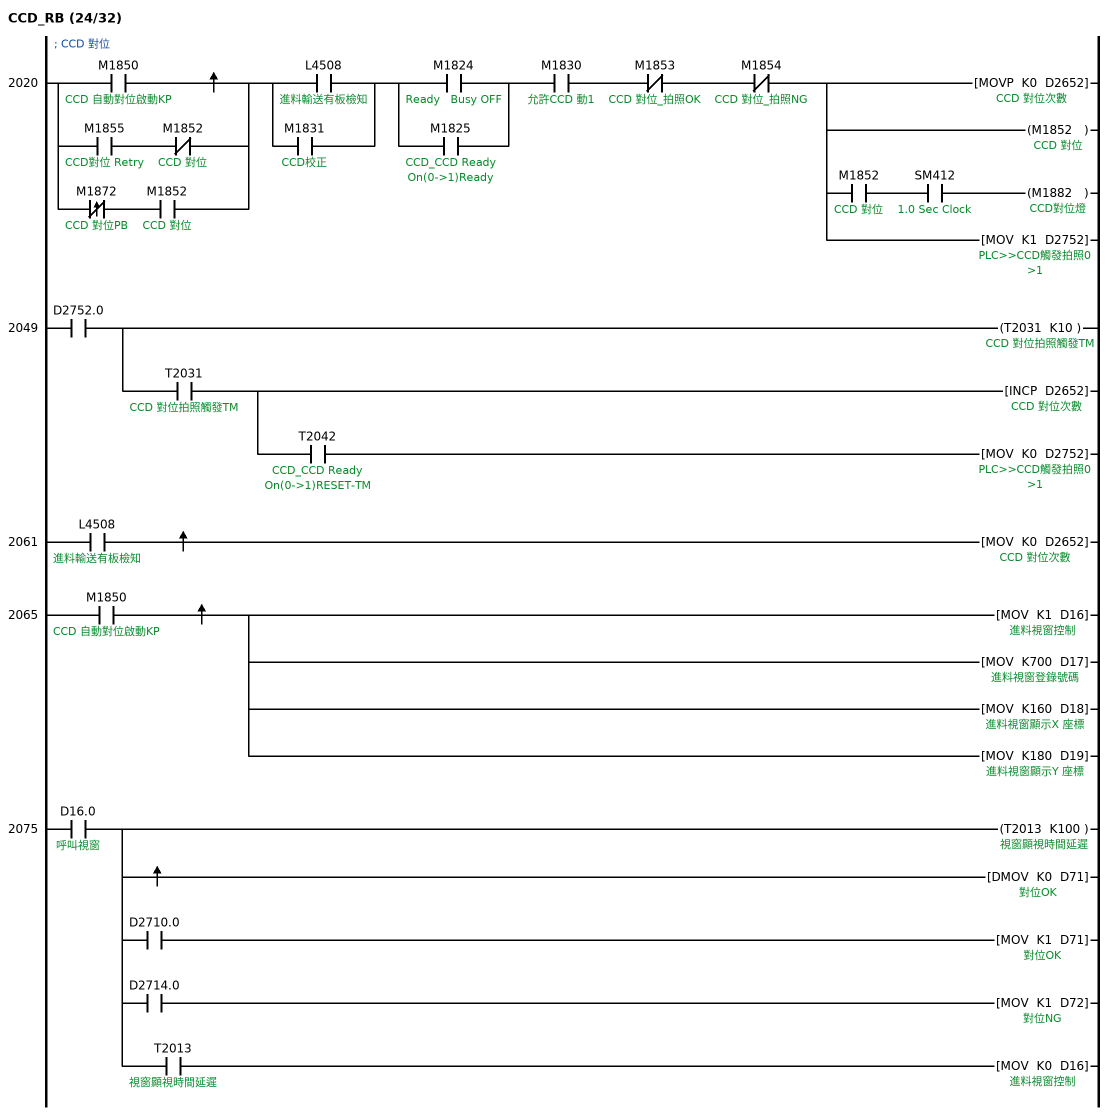
[picture p288: ladder of CCD_RB, rungs at steps 2020 to 2075]
; CCD 對位
2020  LD      M1850  ; CCD 自動對位啟動KP
      MEP
      LD      M1855  ; CCD對位 Retry
      ANI     M1852  ; CCD 對位
      ORB
      LDPI    M1872  ; CCD 對位PB
      AND     M1852  ; CCD 對位
      ORB
      LD      L4508  ; 進料輸送有板檢知
      OR      M1831  ; CCD校正
      ANB
      LD      M1824  ; Ready   Busy OFF
      OR      M1825  ; CCD_CCD Ready On(0->1)Ready
      ANB
      AND     M1830  ; 允許CCD 動1
      ANI     M1853  ; CCD 對位_拍照OK
      ANI     M1854  ; CCD 對位_拍照NG
      MOVP    K0 D2652  ; CCD 對位次數
      OUT     M1852  ; CCD 對位
      MPS
      AND     M1852  ; CCD 對位
      AND     SM412  ; 1.0 Sec Clock
      OUT     M1882  ; CCD對位燈
      MPP
      MOV     K1 D2752
2049  LD      D2752.0
      OUT     T2031 K10  ; CCD 對位拍照觸發TM
      AND     T2031  ; CCD 對位拍照觸發TM
      INCP    D2652
      AND     T2042  ; CCD_CCD Ready On(0->1)RESET-TM
      MOV     K0 D2752
2061  LD      L4508  ; 進料輸送有板檢知
      MEP
      MOV     K0 D2652
2065  LD      M1850  ; CCD 自動對位啟動KP
      MEP
      MOV     K1 D16  ; 進料視窗控制
      MOV     K700 D17  ; 進料視窗登錄號碼
      MOV     K160 D18  ; 進料視窗顯示X 座標
      MOV     K180 D19  ; 進料視窗顯示Y 座標
2075  LD      D16.0  ; 呼叫視窗
      OUT     T2013 K100  ; 視窗顯視時間延遲
      MPS
      MEP
      DMOV    K0 D71  ; 對位OK
      MRD
      AND     D2710.0
      MOV     K1 D71
      MRD
      AND     D2714.0
      MOV     K1 D72  ; 對位NG
      MPP
      AND     T2013  ; 視窗顯視時間延遲
      MOV     K0 D16
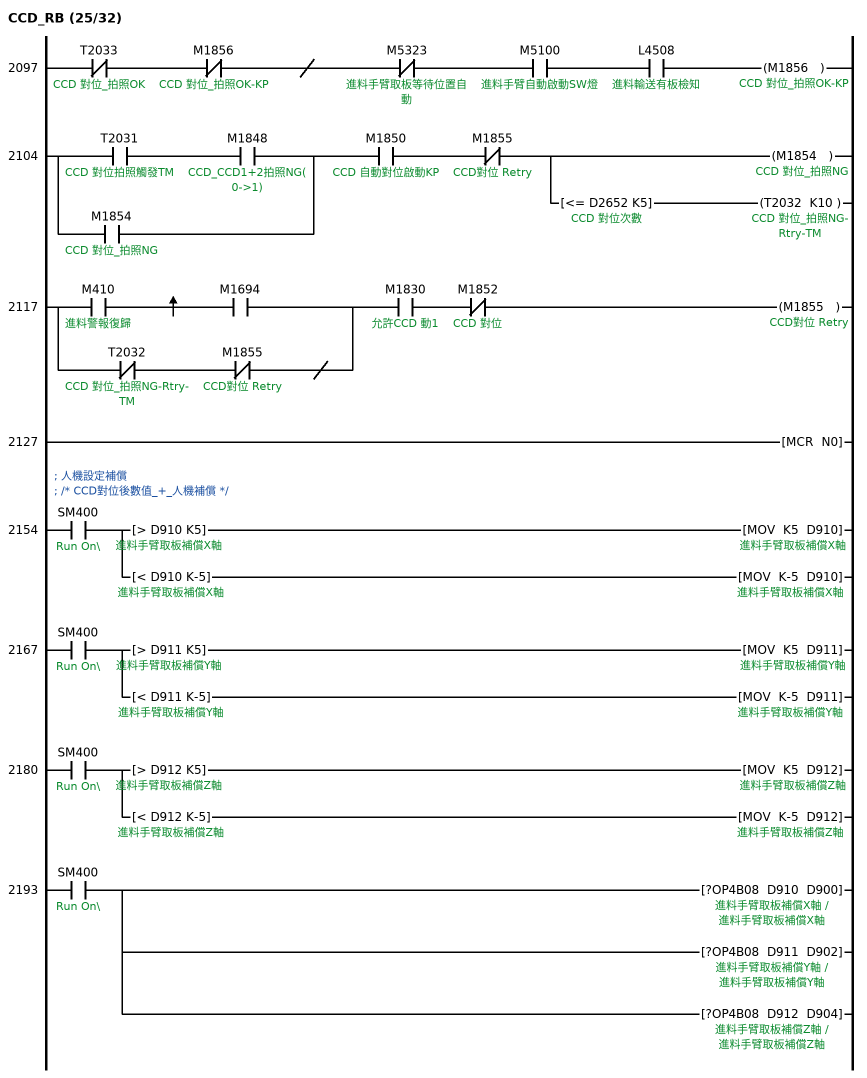
2097  LDI     T2033  ; CCD 對位_拍照OK
      ANI     M1856  ; CCD 對位_拍照OK-KP
      INV
      ANI     M5323  ; 進料手臂取板等待位置自動
      AND     M5100  ; 進料手臂自動啟動SW燈
      AND     L4508  ; 進料輸送有板檢知
      OUT     M1856  ; CCD 對位_拍照OK-KP
2104  LD      T2031  ; CCD 對位拍照觸發TM
      AND     M1848  ; CCD_CCD1+2拍照NG(0->1)
      OR      M1854  ; CCD 對位_拍照NG
      AND     M1850  ; CCD 自動對位啟動KP
      ANI     M1855  ; CCD對位 Retry
      OUT     M1854  ; CCD 對位_拍照NG
      AND<=   D2652 K5  ; CCD 對位次數
      OUT     T2032 K10  ; CCD 對位_拍照NG-Rtry-TM
2117  LD      M410  ; 進料警報復歸
      MEP
      AND     M1694
      LDI     T2032  ; CCD 對位_拍照NG-Rtry-TM
      ANI     M1855  ; CCD對位 Retry
      INV
      ORB
      AND     M1830  ; 允許CCD 動1
      ANI     M1852  ; CCD 對位
      OUT     M1855  ; CCD對位 Retry
2127  MCR     N0
; 人機設定補償
; /* CCD對位後數值_+_人機補償 */
2154  LD      SM400  ; Run On\
      MPS
      AND>    D910 K5  ; 進料手臂取板補償X軸
      MOV     K5 D910
      MPP
      AND<    D910 K-5  ; 進料手臂取板補償X軸
      MOV     K-5 D910
2167  LD      SM400  ; Run On\
      MPS
      AND>    D911 K5  ; 進料手臂取板補償Y軸
      MOV     K5 D911
      MPP
      AND<    D911 K-5  ; 進料手臂取板補償Y軸
      MOV     K-5 D911
2180  LD      SM400  ; Run On\
      MPS
      AND>    D912 K5  ; 進料手臂取板補償Z軸
      MOV     K5 D912
      MPP
      AND<    D912 K-5  ; 進料手臂取板補償Z軸
      MOV     K-5 D912
2193  LD      SM400  ; Run On\
      ?OP4B08 D910 D900  ; 進料手臂取板補償X軸
      ?OP4B08 D911 D902  ; 進料手臂取板補償Y軸
      ?OP4B08 D912 D904  ; 進料手臂取板補償Z軸
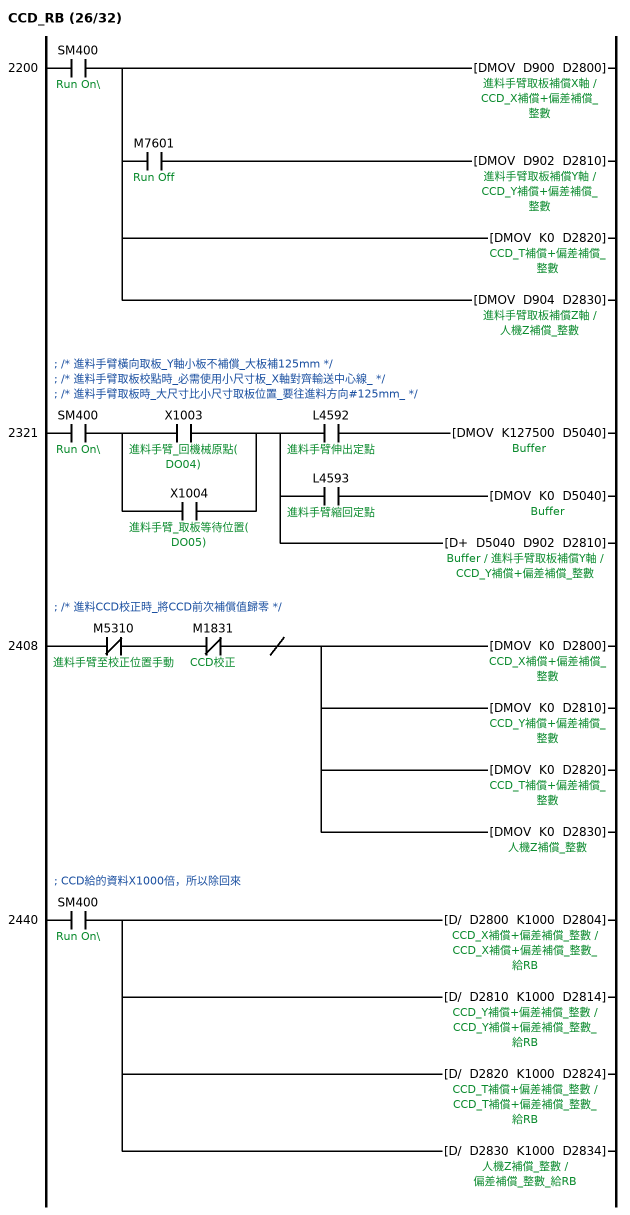
2200  LD      SM400  ; Run On\
      DMOV    D900 D2800  ; CCD_X補償+偏差補償_整數
      MPS
      AND     M7601  ; Run Off
      DMOV    D902 D2810  ; CCD_Y補償+偏差補償_整數
        [note] /* 在大/小板寬已補償位置_ */
      MPP
      DMOV    K0 D2820  ; CCD_T補償+偏差補償_整數
      DMOV    D904 D2830  ; 人機Z補償_整數
; /* 進料手臂橫向取板_Y軸小板不補償_大板補125mm */
; /* 進料手臂取板校點時_必需使用小尺寸板_X軸對齊輸送中心線_ */
; /* 進料手臂取板時_大尺寸比小尺寸取板位置_要往進料方向#125mm_ */
2321  LD      SM400  ; Run On\
      LD      X1003  ; 進料手臂_回機械原點(DO04)
      OR      X1004  ; 進料手臂_取板等待位置(DO05)
      ANB
      MPS
      AND     L4592  ; 進料手臂伸出定點
      DMOV    K127500 D5040  ; Buffer
        [note] /* 手臂大板寬_取板位_SHIFT */
      MRD
      AND     L4593  ; 進料手臂縮回定點
      DMOV    K0 D5040
        [note] /* 手臂大板寬_取板位_SHIFT */
      MPP
      D+      D5040 D902 D2810
        [note] /* 人機設定補正板長 */
; /* 進料CCD校正時_將CCD前次補償值歸零 */
2408  LDI     M5310  ; 進料手臂至校正位置手動
      ANI     M1831  ; CCD校正
      INV
      DMOV    K0 D2800
      DMOV    K0 D2810
      DMOV    K0 D2820
      DMOV    K0 D2830
; CCD給的資料X1000倍，所以除回來
2440  LD      SM400  ; Run On\
      D/      D2800 K1000 D2804
      D/      D2810 K1000 D2814
      D/      D2820 K1000 D2824
      D/      D2830 K1000 D2834  ; 偏差補償_整數_給RB
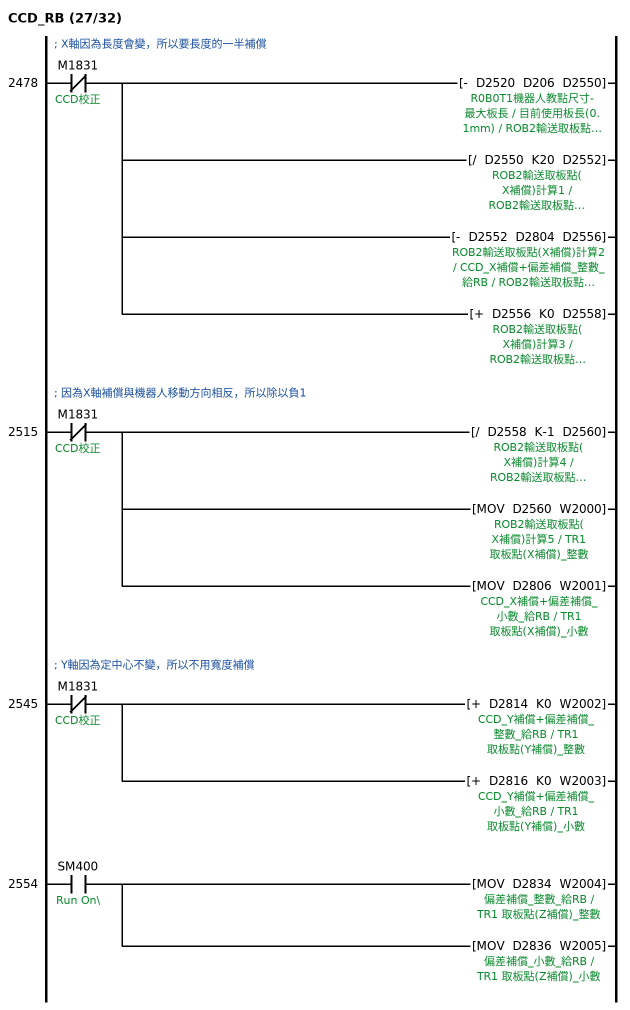
; X軸因為長度會變，所以要長度的一半補償
2478  LDI     M1831  ; CCD校正
      -       D2520 D206 D2550  ; R0B0T1機器人教點尺寸-最大板長 / 目前使用板長(0.1mm) / ROB2輸送取板點(X補償)計算1
      /       D2550 K20 D2552  ; ROB2輸送取板點(X補償)計算2
      -       D2552 D2804 D2556  ; ROB2輸送取板點(X補償)計算3
      +       D2556 K0 D2558  ; ROB2輸送取板點(X補償)計算4
; 因為X軸補償與機器人移動方向相反，所以除以負1
2515  LDI     M1831  ; CCD校正
      /       D2558 K-1 D2560  ; ROB2輸送取板點(X補償)計算5
      MOV     D2560 W2000  ; TR1 取板點(X補償)_整數
      MOV     D2806 W2001  ; CCD_X補償+偏差補償_小數_給RB / TR1 取板點(X補償)_小數
; Y軸因為定中心不變，所以不用寬度補償
2545  LDI     M1831  ; CCD校正
      +       D2814 K0 W2002  ; TR1 取板點(Y補償)_整數
      +       D2816 K0 W2003  ; CCD_Y補償+偏差補償_小數_給RB / TR1 取板點(Y補償)_小數
2554  LD      SM400  ; Run On\
      MOV     D2834 W2004  ; TR1 取板點(Z補償)_整數
      MOV     D2836 W2005  ; 偏差補償_小數_給RB / TR1 取板點(Z補償)_小數
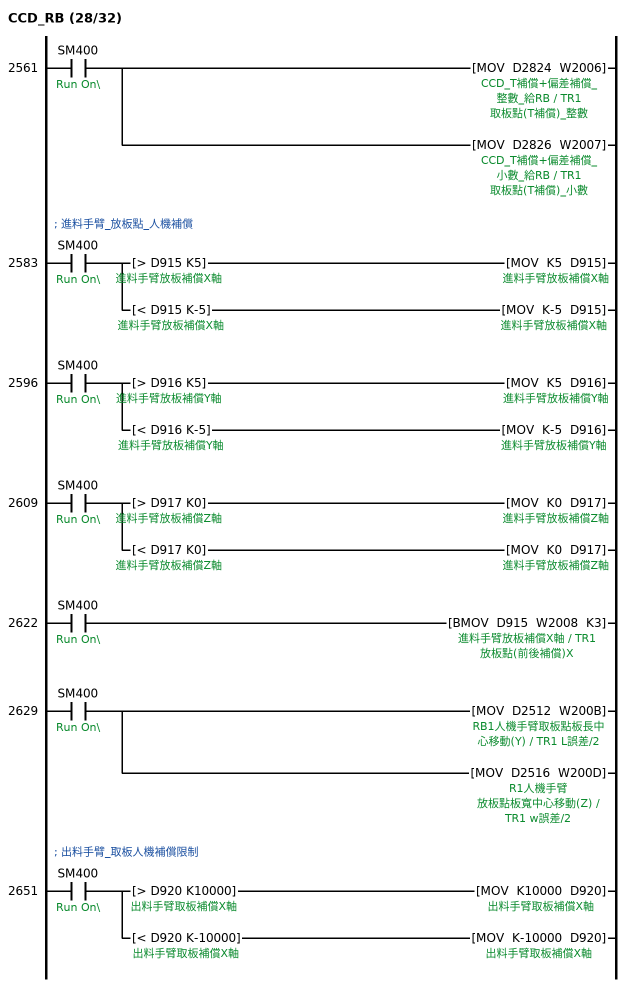
2561  LD      SM400  ; Run On\
      MOV     D2824 W2006  ; TR1 取板點(T補償)_整數
      MOV     D2826 W2007  ; CCD_T補償+偏差補償_小數_給RB / TR1 取板點(T補償)_小數
; 進料手臂_放板點_人機補償
2583  LD      SM400  ; Run On\
      MPS
      AND>    D915 K5  ; 進料手臂放板補償X軸
      MOV     K5 D915
      MPP
      AND<    D915 K-5  ; 進料手臂放板補償X軸
      MOV     K-5 D915
2596  LD      SM400  ; Run On\
      MPS
      AND>    D916 K5  ; 進料手臂放板補償Y軸
      MOV     K5 D916
      MPP
      AND<    D916 K-5  ; 進料手臂放板補償Y軸
      MOV     K-5 D916
2609  LD      SM400  ; Run On\
      MPS
      AND>    D917 K0  ; 進料手臂放板補償Z軸
      MOV     K0 D917
      MPP
      AND<    D917 K0  ; 進料手臂放板補償Z軸
      MOV     K0 D917
2622  LD      SM400  ; Run On\
      BMOV    D915 W2008 K3  ; TR1 放板點(前後補償)X
2629  LD      SM400  ; Run On\
      MOV     D2512 W200B  ; RB1人機手臂取板點板長中心移動(Y) / TR1 L誤差/2
      MOV     D2516 W200D  ; R1人機手臂 放板點板寬中心移動(Z) / TR1 w誤差/2
; 出料手臂_取板人機補償限制
2651  LD      SM400  ; Run On\
      MPS
      AND>    D920 K10000  ; 出料手臂取板補償X軸
      MOV     K10000 D920
      MPP
      AND<    D920 K-10000  ; 出料手臂取板補償X軸
      MOV     K-10000 D920
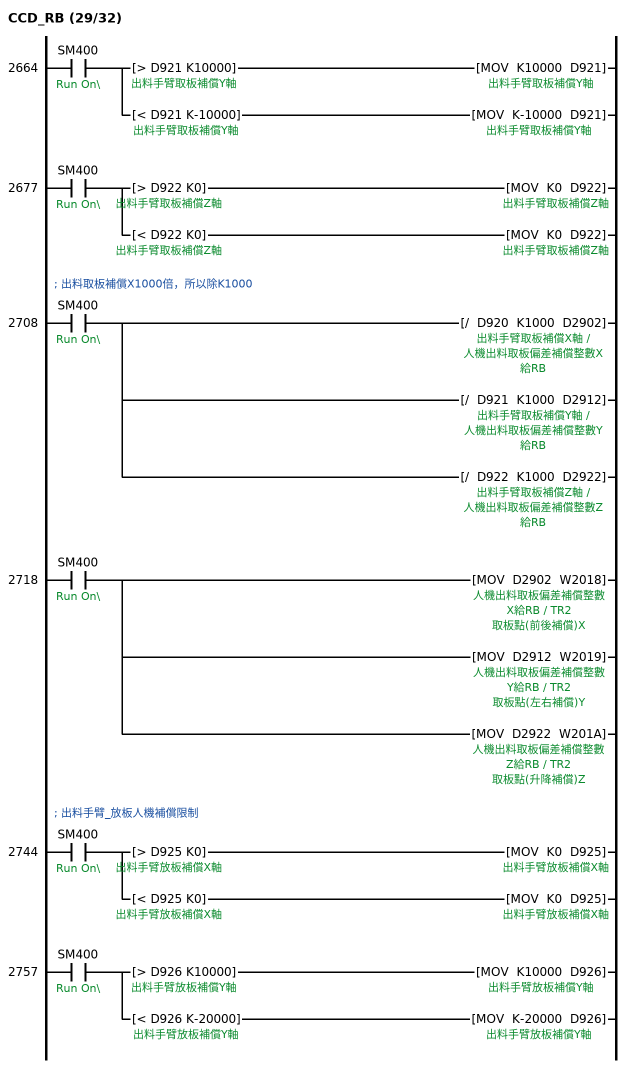
2664  LD      SM400  ; Run On\
      MPS
      AND>    D921 K10000  ; 出料手臂取板補償Y軸
      MOV     K10000 D921
      MPP
      AND<    D921 K-10000  ; 出料手臂取板補償Y軸
      MOV     K-10000 D921
2677  LD      SM400  ; Run On\
      MPS
      AND>    D922 K0  ; 出料手臂取板補償Z軸
      MOV     K0 D922
      MPP
      AND<    D922 K0  ; 出料手臂取板補償Z軸
      MOV     K0 D922
; 出料取板補償X1000倍，所以除K1000
2708  LD      SM400  ; Run On\
      /       D920 K1000 D2902  ; 人機出料取板偏差補償整數X給RB
      /       D921 K1000 D2912  ; 人機出料取板偏差補償整數Y給RB
      /       D922 K1000 D2922  ; 人機出料取板偏差補償整數Z給RB
2718  LD      SM400  ; Run On\
      MOV     D2902 W2018  ; TR2 取板點(前後補償)X
      MOV     D2912 W2019  ; TR2 取板點(左右補償)Y
      MOV     D2922 W201A  ; TR2 取板點(升降補償)Z
; 出料手臂_放板人機補償限制
2744  LD      SM400  ; Run On\
      MPS
      AND>    D925 K0  ; 出料手臂放板補償X軸
      MOV     K0 D925
      MPP
      AND<    D925 K0  ; 出料手臂放板補償X軸
      MOV     K0 D925
2757  LD      SM400  ; Run On\
      MPS
      AND>    D926 K10000  ; 出料手臂放板補償Y軸
      MOV     K10000 D926
      MPP
      AND<    D926 K-20000  ; 出料手臂放板補償Y軸
      MOV     K-20000 D926
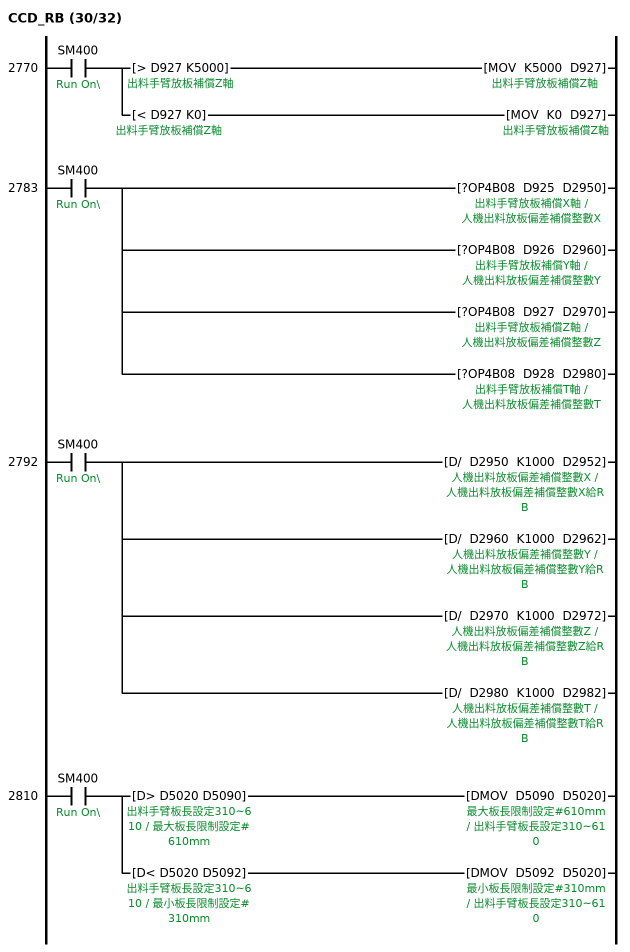
2770  LD      SM400  ; Run On\
      MPS
      AND>    D927 K5000  ; 出料手臂放板補償Z軸
      MOV     K5000 D927
      MPP
      AND<    D927 K0  ; 出料手臂放板補償Z軸
      MOV     K0 D927
2783  LD      SM400  ; Run On\
      ?OP4B08 D925 D2950  ; 人機出料放板偏差補償整數X
      ?OP4B08 D926 D2960  ; 人機出料放板偏差補償整數Y
      ?OP4B08 D927 D2970  ; 人機出料放板偏差補償整數Z
      ?OP4B08 D928 D2980  ; 出料手臂放板補償T軸 / 人機出料放板偏差補償整數T
2792  LD      SM400  ; Run On\
      D/      D2950 K1000 D2952  ; 人機出料放板偏差補償整數X給RB
      D/      D2960 K1000 D2962  ; 人機出料放板偏差補償整數Y給RB
      D/      D2970 K1000 D2972  ; 人機出料放板偏差補償整數Z給RB
      D/      D2980 K1000 D2982  ; 人機出料放板偏差補償整數T給RB
2810  LD      SM400  ; Run On\
      MPS
      ANDD>   D5020 D5090  ; 出料手臂板長設定310~610 / 最大板長限制設定#610mm
      DMOV    D5090 D5020
      MPP
      ANDD<   D5020 D5092  ; 出料手臂板長設定310~610 / 最小板長限制設定#310mm
      DMOV    D5092 D5020
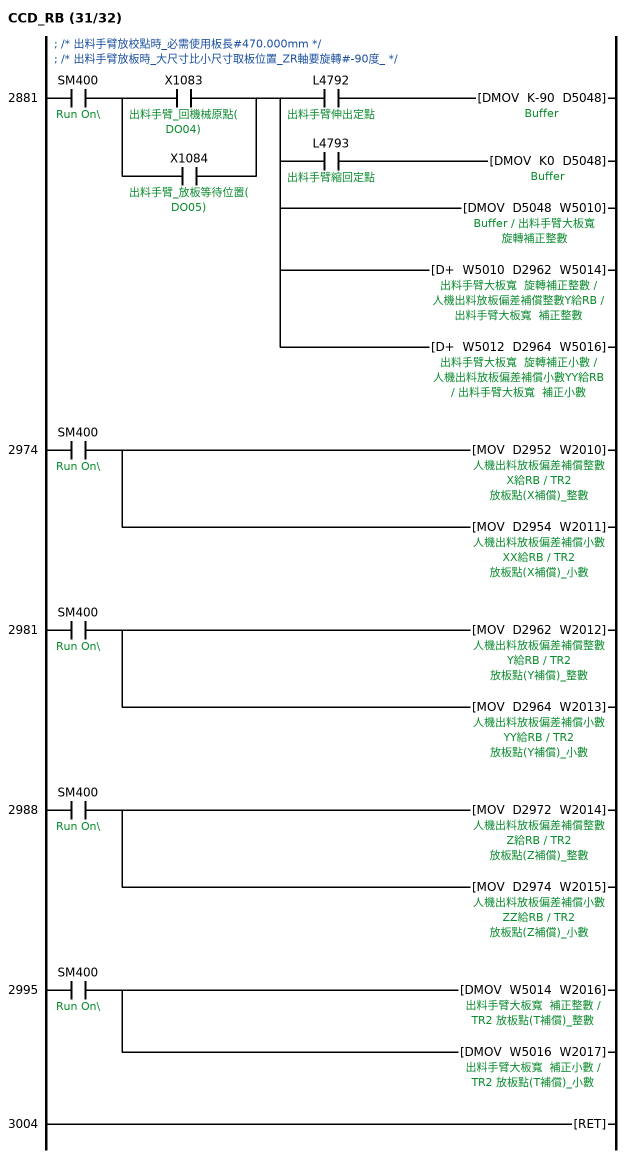
; /* 出料手臂放校點時_必需使用板長#470.000mm */
; /* 出料手臂放板時_大尺寸比小尺寸取板位置_ZR軸要旋轉#-90度_ */
2881  LD      SM400  ; Run On\
      LD      X1083  ; 出料手臂_回機械原點(DO04)
      OR      X1084  ; 出料手臂_放板等待位置(DO05)
      ANB
      MPS
      AND     L4792  ; 出料手臂伸出定點
      DMOV    K-90 D5048  ; Buffer
        [note] /* 手臂大板寬_取板位_SHIFT */
      MRD
      AND     L4793  ; 出料手臂縮回定點
      DMOV    K0 D5048
        [note] /* 手臂大板寬_取板位_SHIFT */
      MPP
      DMOV    D5048 W5010  ; 出料手臂大板寬  旋轉補正整數
      D+      W5010 D2962 W5014  ; 出料手臂大板寬  補正整數
        [note] /* 人機設定補正板長整數 */
      D+      W5012 D2964 W5016  ; 出料手臂大板寬  旋轉補正小數 / 人機出料放板偏差補償小數YY給RB / 出料手臂大板寬  補正小數
        [note] /* 人機設定補正板長小數 */
2974  LD      SM400  ; Run On\
      MOV     D2952 W2010  ; TR2 放板點(X補償)_整數
      MOV     D2954 W2011  ; 人機出料放板偏差補償小數XX給RB / TR2 放板點(X補償)_小數
2981  LD      SM400  ; Run On\
      MOV     D2962 W2012  ; TR2 放板點(Y補償)_整數
      MOV     D2964 W2013  ; TR2 放板點(Y補償)_小數
2988  LD      SM400  ; Run On\
      MOV     D2972 W2014  ; TR2 放板點(Z補償)_整數
      MOV     D2974 W2015  ; 人機出料放板偏差補償小數ZZ給RB / TR2 放板點(Z補償)_小數
2995  LD      SM400  ; Run On\
      DMOV    W5014 W2016  ; TR2 放板點(T補償)_整數
      DMOV    W5016 W2017  ; TR2 放板點(T補償)_小數
3004  RET
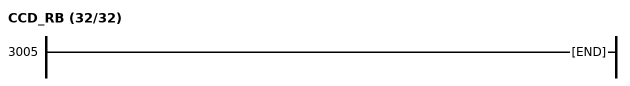
3005  END
END_PROGRAM

PROGRAM MECHA
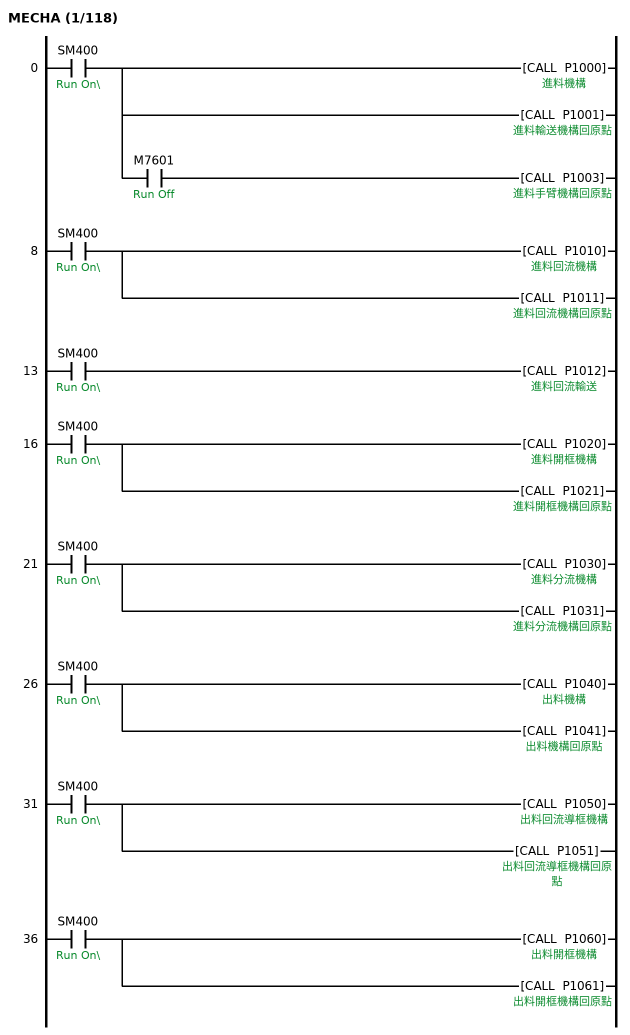
0     LD      SM400  ; Run On\
      CALL    P1000  ; 進料機構
      CALL    P1001  ; 進料輸送機構回原點
      AND     M7601  ; Run Off
      CALL    P1003  ; 進料手臂機構回原點
8     LD      SM400  ; Run On\
      CALL    P1010  ; 進料回流機構
      CALL    P1011  ; 進料回流機構回原點
13    LD      SM400  ; Run On\
      CALL    P1012  ; 進料回流輸送
16    LD      SM400  ; Run On\
      CALL    P1020  ; 進料開框機構
      CALL    P1021  ; 進料開框機構回原點
21    LD      SM400  ; Run On\
      CALL    P1030  ; 進料分流機構
      CALL    P1031  ; 進料分流機構回原點
26    LD      SM400  ; Run On\
      CALL    P1040  ; 出料機構
      CALL    P1041  ; 出料機構回原點
31    LD      SM400  ; Run On\
      CALL    P1050  ; 出料回流導框機構
      CALL    P1051  ; 出料回流導框機構回原點
36    LD      SM400  ; Run On\
      CALL    P1060  ; 出料開框機構
      CALL    P1061  ; 出料開框機構回原點
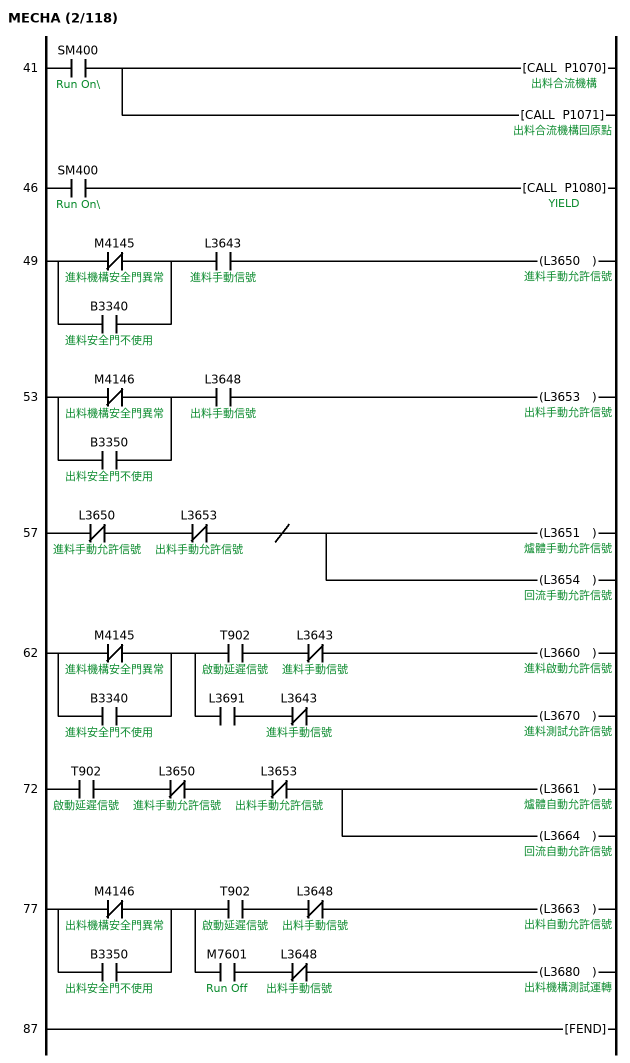
41    LD      SM400  ; Run On\
      CALL    P1070  ; 出料合流機構
      CALL    P1071  ; 出料合流機構回原點
46    LD      SM400  ; Run On\
      CALL    P1080  ; YIELD
49    LDI     M4145  ; 進料機構安全門異常
      OR      B3340  ; 進料安全門不使用
      AND     L3643  ; 進料手動信號
      OUT     L3650  ; 進料手動允許信號
53    LDI     M4146  ; 出料機構安全門異常
      OR      B3350  ; 出料安全門不使用
      AND     L3648  ; 出料手動信號
      OUT     L3653  ; 出料手動允許信號
57    LDI     L3650  ; 進料手動允許信號
      ANI     L3653  ; 出料手動允許信號
      INV
      OUT     L3651  ; 爐體手動允許信號
      OUT     L3654  ; 回流手動允許信號
62    LDI     M4145  ; 進料機構安全門異常
      OR      B3340  ; 進料安全門不使用
      MPS
      AND     T902  ; 啟動延遲信號
      ANI     L3643  ; 進料手動信號
      OUT     L3660  ; 進料啟動允許信號
      MPP
      AND     L3691
      ANI     L3643  ; 進料手動信號
      OUT     L3670  ; 進料測試允許信號
72    LD      T902  ; 啟動延遲信號
      ANI     L3650  ; 進料手動允許信號
      ANI     L3653  ; 出料手動允許信號
      OUT     L3661  ; 爐體自動允許信號
      OUT     L3664  ; 回流自動允許信號
77    LDI     M4146  ; 出料機構安全門異常
      OR      B3350  ; 出料安全門不使用
      MPS
      AND     T902  ; 啟動延遲信號
      ANI     L3648  ; 出料手動信號
      OUT     L3663  ; 出料自動允許信號
      MPP
      AND     M7601  ; Run Off
      ANI     L3648  ; 出料手動信號
      OUT     L3680  ; 出料機構測試運轉
87    FEND
; ---------進料機構------
      P1000
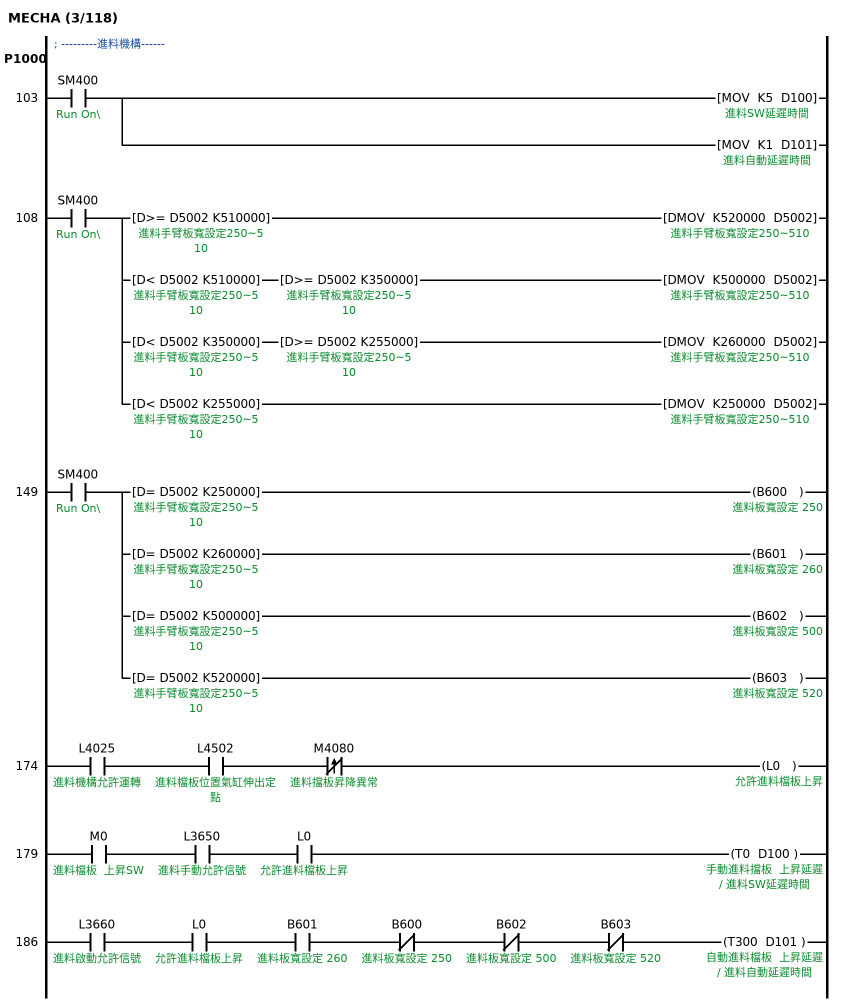
103   LD      SM400  ; Run On\
      MOV     K5 D100  ; 進料SW延遲時間
      MOV     K1 D101  ; 進料自動延遲時間
108   LD      SM400  ; Run On\
      MPS
      ANDD>=  D5002 K510000  ; 進料手臂板寬設定250~510
      DMOV    K520000 D5002
      MRD
      ANDD<   D5002 K510000  ; 進料手臂板寬設定250~510
      ANDD>=  D5002 K350000  ; 進料手臂板寬設定250~510
      DMOV    K500000 D5002
      MRD
      ANDD<   D5002 K350000  ; 進料手臂板寬設定250~510
      ANDD>=  D5002 K255000  ; 進料手臂板寬設定250~510
      DMOV    K260000 D5002
      MPP
      ANDD<   D5002 K255000  ; 進料手臂板寬設定250~510
      DMOV    K250000 D5002
149   LD      SM400  ; Run On\
      MPS
      ANDD=   D5002 K250000  ; 進料手臂板寬設定250~510
      OUT     B600  ; 進料板寬設定 250
      MRD
      ANDD=   D5002 K260000  ; 進料手臂板寬設定250~510
      OUT     B601  ; 進料板寬設定 260
      MRD
      ANDD=   D5002 K500000  ; 進料手臂板寬設定250~510
      OUT     B602  ; 進料板寬設定 500
      MPP
      ANDD=   D5002 K520000  ; 進料手臂板寬設定250~510
      OUT     B603  ; 進料板寬設定 520
174   LD      L4025  ; 進料機構允許運轉
      AND     L4502  ; 進料檔板位置氣缸伸出定點
      ANDPI   M4080  ; 進料擋板昇降異常
      OUT     L0  ; 允許進料檔板上昇
179   LD      M0  ; 進料檔板  上昇SW
      AND     L3650  ; 進料手動允許信號
      AND     L0  ; 允許進料檔板上昇
      OUT     T0 D100  ; 手動進料擋板  上昇延遲 / 進料SW延遲時間
186   LD      L3660  ; 進料啟動允許信號
      AND     L0  ; 允許進料檔板上昇
      AND     B601  ; 進料板寬設定 260
      ANI     B600  ; 進料板寬設定 250
      ANI     B602  ; 進料板寬設定 500
      ANI     B603  ; 進料板寬設定 520
      OUT     T300 D101  ; 自動進料檔板  上昇延遲 / 進料自動延遲時間
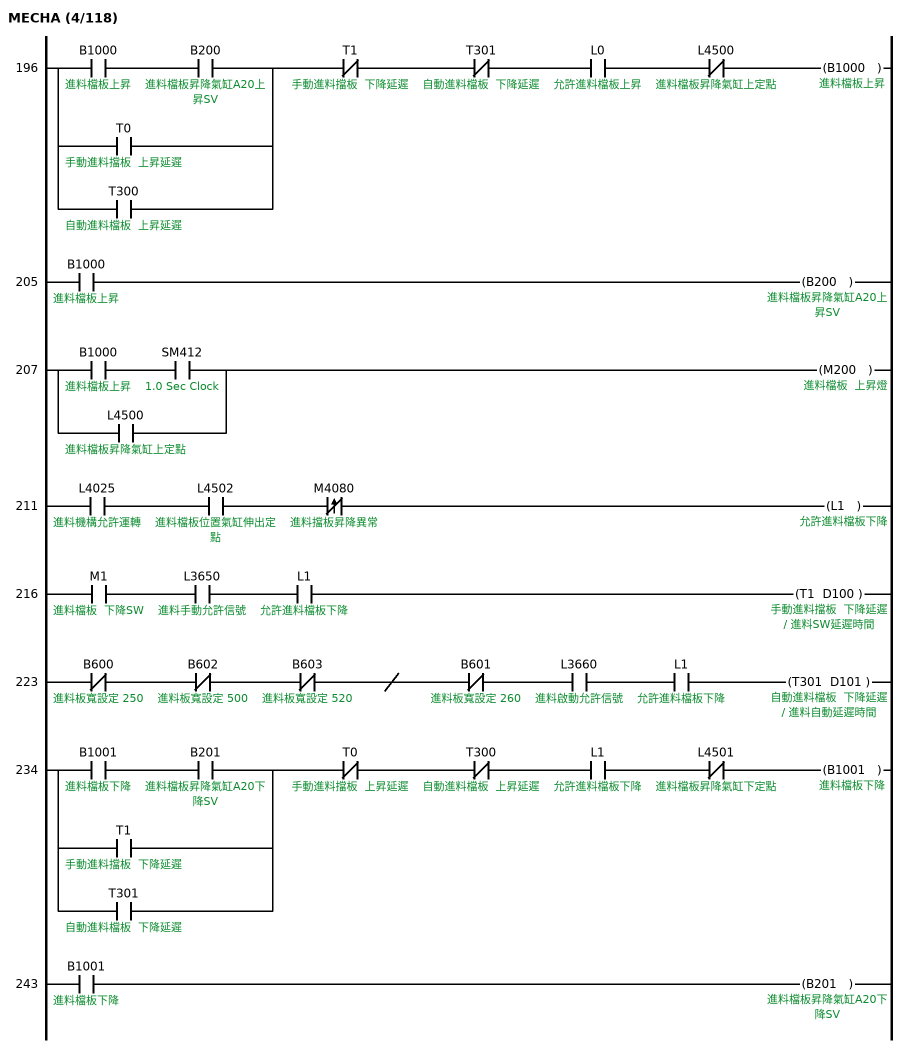
196   LD      B1000  ; 進料檔板上昇
      AND     B200  ; 進料檔板昇降氣缸A20上昇SV
      OR      T0  ; 手動進料擋板  上昇延遲
      OR      T300  ; 自動進料檔板  上昇延遲
      ANI     T1  ; 手動進料擋板  下降延遲
      ANI     T301  ; 自動進料檔板  下降延遲
      AND     L0  ; 允許進料檔板上昇
      ANI     L4500  ; 進料檔板昇降氣缸上定點
      OUT     B1000  ; 進料檔板上昇
205   LD      B1000  ; 進料檔板上昇
      OUT     B200  ; 進料檔板昇降氣缸A20上昇SV
207   LD      B1000  ; 進料檔板上昇
      AND     SM412  ; 1.0 Sec Clock
      OR      L4500  ; 進料檔板昇降氣缸上定點
      OUT     M200  ; 進料檔板  上昇燈
211   LD      L4025  ; 進料機構允許運轉
      AND     L4502  ; 進料檔板位置氣缸伸出定點
      ANDPI   M4080  ; 進料擋板昇降異常
      OUT     L1  ; 允許進料檔板下降
216   LD      M1  ; 進料檔板  下降SW
      AND     L3650  ; 進料手動允許信號
      AND     L1  ; 允許進料檔板下降
      OUT     T1 D100  ; 手動進料擋板  下降延遲 / 進料SW延遲時間
223   LDI     B600  ; 進料板寬設定 250
      ANI     B602  ; 進料板寬設定 500
      ANI     B603  ; 進料板寬設定 520
      INV
      ANI     B601  ; 進料板寬設定 260
      AND     L3660  ; 進料啟動允許信號
      AND     L1  ; 允許進料檔板下降
      OUT     T301 D101  ; 自動進料檔板  下降延遲 / 進料自動延遲時間
234   LD      B1001  ; 進料檔板下降
      AND     B201  ; 進料檔板昇降氣缸A20下降SV
      OR      T1  ; 手動進料擋板  下降延遲
      OR      T301  ; 自動進料檔板  下降延遲
      ANI     T0  ; 手動進料擋板  上昇延遲
      ANI     T300  ; 自動進料檔板  上昇延遲
      AND     L1  ; 允許進料檔板下降
      ANI     L4501  ; 進料檔板昇降氣缸下定點
      OUT     B1001  ; 進料檔板下降
243   LD      B1001  ; 進料檔板下降
      OUT     B201  ; 進料檔板昇降氣缸A20下降SV
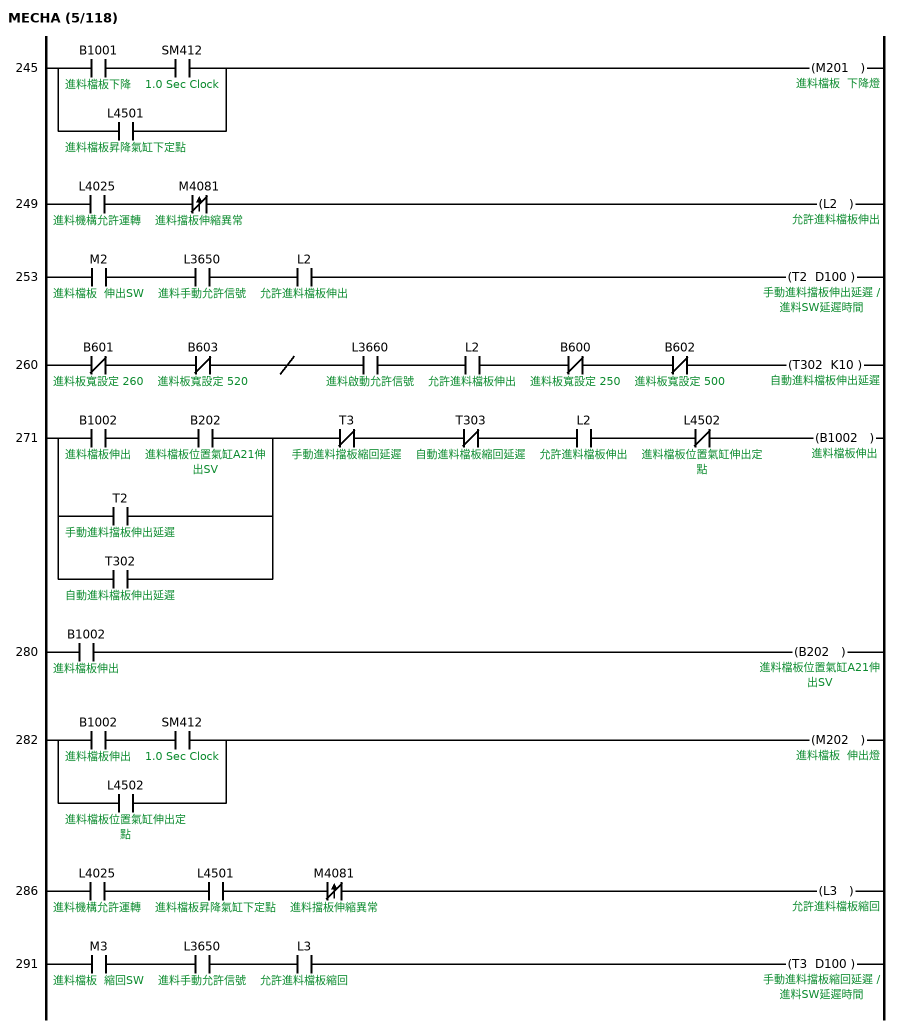
245   LD      B1001  ; 進料檔板下降
      AND     SM412  ; 1.0 Sec Clock
      OR      L4501  ; 進料檔板昇降氣缸下定點
      OUT     M201  ; 進料檔板  下降燈
249   LD      L4025  ; 進料機構允許運轉
      ANDPI   M4081  ; 進料擋板伸縮異常
      OUT     L2  ; 允許進料檔板伸出
253   LD      M2  ; 進料檔板  伸出SW
      AND     L3650  ; 進料手動允許信號
      AND     L2  ; 允許進料檔板伸出
      OUT     T2 D100  ; 手動進料擋板伸出延遲 / 進料SW延遲時間
260   LDI     B601  ; 進料板寬設定 260
      ANI     B603  ; 進料板寬設定 520
      INV
      AND     L3660  ; 進料啟動允許信號
      AND     L2  ; 允許進料檔板伸出
      ANI     B600  ; 進料板寬設定 250
      ANI     B602  ; 進料板寬設定 500
      OUT     T302 K10  ; 自動進料檔板伸出延遲
271   LD      B1002  ; 進料檔板伸出
      AND     B202  ; 進料檔板位置氣缸A21伸出SV
      OR      T2  ; 手動進料擋板伸出延遲
      OR      T302  ; 自動進料檔板伸出延遲
      ANI     T3  ; 手動進料擋板縮回延遲
      ANI     T303  ; 自動進料檔板縮回延遲
      AND     L2  ; 允許進料檔板伸出
      ANI     L4502  ; 進料檔板位置氣缸伸出定點
      OUT     B1002  ; 進料檔板伸出
280   LD      B1002  ; 進料檔板伸出
      OUT     B202  ; 進料檔板位置氣缸A21伸出SV
282   LD      B1002  ; 進料檔板伸出
      AND     SM412  ; 1.0 Sec Clock
      OR      L4502  ; 進料檔板位置氣缸伸出定點
      OUT     M202  ; 進料檔板  伸出燈
286   LD      L4025  ; 進料機構允許運轉
      AND     L4501  ; 進料檔板昇降氣缸下定點
      ANDPI   M4081  ; 進料擋板伸縮異常
      OUT     L3  ; 允許進料檔板縮回
291   LD      M3  ; 進料檔板  縮回SW
      AND     L3650  ; 進料手動允許信號
      AND     L3  ; 允許進料檔板縮回
      OUT     T3 D100  ; 手動進料擋板縮回延遲 / 進料SW延遲時間
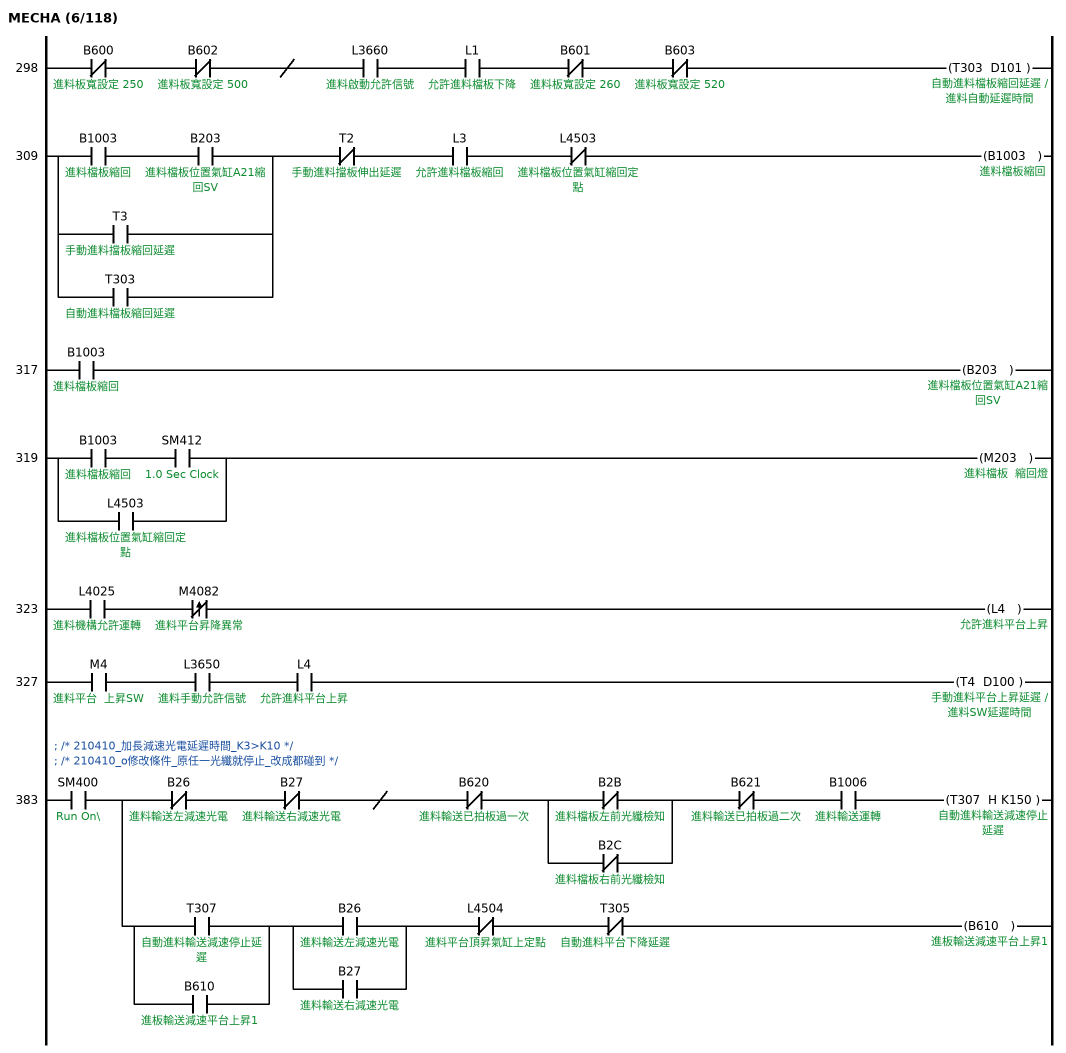
298   LDI     B600  ; 進料板寬設定 250
      ANI     B602  ; 進料板寬設定 500
      INV
      AND     L3660  ; 進料啟動允許信號
      AND     L1  ; 允許進料檔板下降
      ANI     B601  ; 進料板寬設定 260
      ANI     B603  ; 進料板寬設定 520
      OUT     T303 D101  ; 自動進料檔板縮回延遲 / 進料自動延遲時間
309   LD      B1003  ; 進料檔板縮回
      AND     B203  ; 進料檔板位置氣缸A21縮回SV
      OR      T3  ; 手動進料擋板縮回延遲
      OR      T303  ; 自動進料檔板縮回延遲
      ANI     T2  ; 手動進料擋板伸出延遲
      AND     L3  ; 允許進料檔板縮回
      ANI     L4503  ; 進料檔板位置氣缸縮回定點
      OUT     B1003  ; 進料檔板縮回
317   LD      B1003  ; 進料檔板縮回
      OUT     B203  ; 進料檔板位置氣缸A21縮回SV
319   LD      B1003  ; 進料檔板縮回
      AND     SM412  ; 1.0 Sec Clock
      OR      L4503  ; 進料檔板位置氣缸縮回定點
      OUT     M203  ; 進料檔板  縮回燈
323   LD      L4025  ; 進料機構允許運轉
      ANDPI   M4082  ; 進料平台昇降異常
      OUT     L4  ; 允許進料平台上昇
327   LD      M4  ; 進料平台  上昇SW
      AND     L3650  ; 進料手動允許信號
      AND     L4  ; 允許進料平台上昇
      OUT     T4 D100  ; 手動進料平台上昇延遲 / 進料SW延遲時間
; /* 210410_加長減速光電延遲時間_K3>K10 */
; /* 210410_o修改條件_原任一光纖就停止_改成都碰到 */
383   LD      SM400  ; Run On\
      MPS
      ANI     B26  ; 進料輸送左減速光電
      ANI     B27  ; 進料輸送右減速光電
      INV
      ANI     B620  ; 進料輸送已拍板過一次
      LDI     B2B  ; 進料檔板左前光纖檢知
      ORI     B2C  ; 進料檔板右前光纖檢知
      ANB
      ANI     B621  ; 進料輸送已拍板過二次
      AND     B1006  ; 進料輸送運轉
      OUTH    T307 K150  ; 自動進料輸送減速停止延遲
      MPP
      LD      T307  ; 自動進料輸送減速停止延遲
      OR      B610  ; 進板輸送減速平台上昇1
      ANB
      LD      B26  ; 進料輸送左減速光電
      OR      B27  ; 進料輸送右減速光電
      ANB
      ANI     L4504  ; 進料平台頂昇氣缸上定點
      ANI     T305  ; 自動進料平台下降延遲
      OUT     B610  ; 進板輸送減速平台上昇1
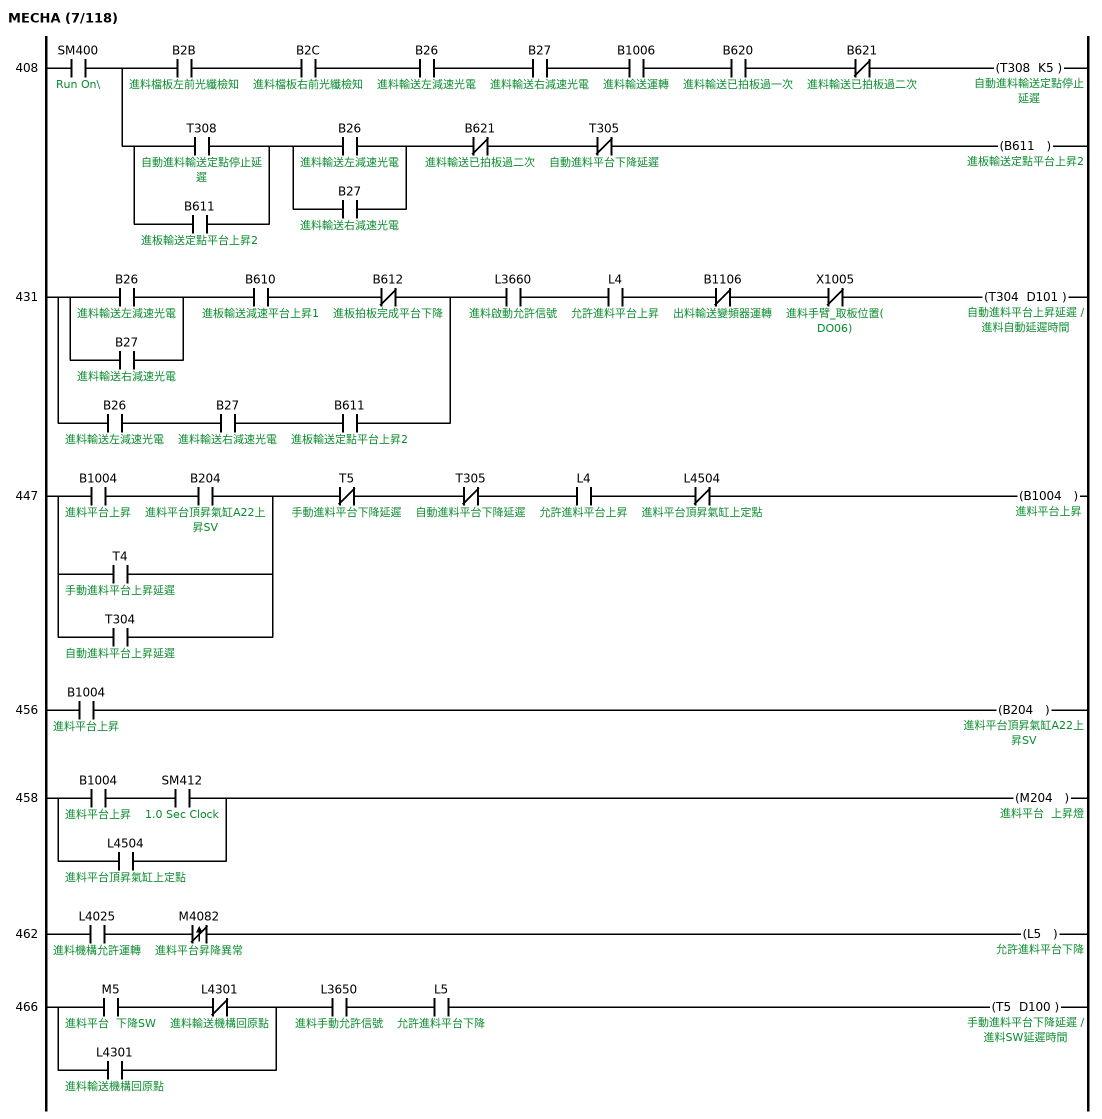
408   LD      SM400  ; Run On\
      MPS
      AND     B2B  ; 進料檔板左前光纖檢知
      AND     B2C  ; 進料檔板右前光纖檢知
      AND     B26  ; 進料輸送左減速光電
      AND     B27  ; 進料輸送右減速光電
      AND     B1006  ; 進料輸送運轉
      AND     B620  ; 進料輸送已拍板過一次
      ANI     B621  ; 進料輸送已拍板過二次
      OUT     T308 K5  ; 自動進料輸送定點停止延遲
      MPP
      LD      T308  ; 自動進料輸送定點停止延遲
      OR      B611  ; 進板輸送定點平台上昇2
      ANB
      LD      B26  ; 進料輸送左減速光電
      OR      B27  ; 進料輸送右減速光電
      ANB
      ANI     B621  ; 進料輸送已拍板過二次
      ANI     T305  ; 自動進料平台下降延遲
      OUT     B611  ; 進板輸送定點平台上昇2
431   LD      B26  ; 進料輸送左減速光電
      OR      B27  ; 進料輸送右減速光電
      AND     B610  ; 進板輸送減速平台上昇1
      ANI     B612  ; 進板拍板完成平台下降
      LD      B26  ; 進料輸送左減速光電
      AND     B27  ; 進料輸送右減速光電
      AND     B611  ; 進板輸送定點平台上昇2
      ORB
      AND     L3660  ; 進料啟動允許信號
      AND     L4  ; 允許進料平台上昇
      ANI     B1106  ; 出料輸送變頻器運轉
      ANI     X1005  ; 進料手臂_取板位置(DO06)
      OUT     T304 D101  ; 自動進料平台上昇延遲 / 進料自動延遲時間
447   LD      B1004  ; 進料平台上昇
      AND     B204  ; 進料平台頂昇氣缸A22上昇SV
      OR      T4  ; 手動進料平台上昇延遲
      OR      T304  ; 自動進料平台上昇延遲
      ANI     T5  ; 手動進料平台下降延遲
      ANI     T305  ; 自動進料平台下降延遲
      AND     L4  ; 允許進料平台上昇
      ANI     L4504  ; 進料平台頂昇氣缸上定點
      OUT     B1004  ; 進料平台上昇
456   LD      B1004  ; 進料平台上昇
      OUT     B204  ; 進料平台頂昇氣缸A22上昇SV
458   LD      B1004  ; 進料平台上昇
      AND     SM412  ; 1.0 Sec Clock
      OR      L4504  ; 進料平台頂昇氣缸上定點
      OUT     M204  ; 進料平台  上昇燈
462   LD      L4025  ; 進料機構允許運轉
      ANDPI   M4082  ; 進料平台昇降異常
      OUT     L5  ; 允許進料平台下降
466   LD      M5  ; 進料平台  下降SW
      ANI     L4301  ; 進料輸送機構回原點
      OR      L4301  ; 進料輸送機構回原點
      AND     L3650  ; 進料手動允許信號
      AND     L5  ; 允許進料平台下降
      OUT     T5 D100  ; 手動進料平台下降延遲 / 進料SW延遲時間
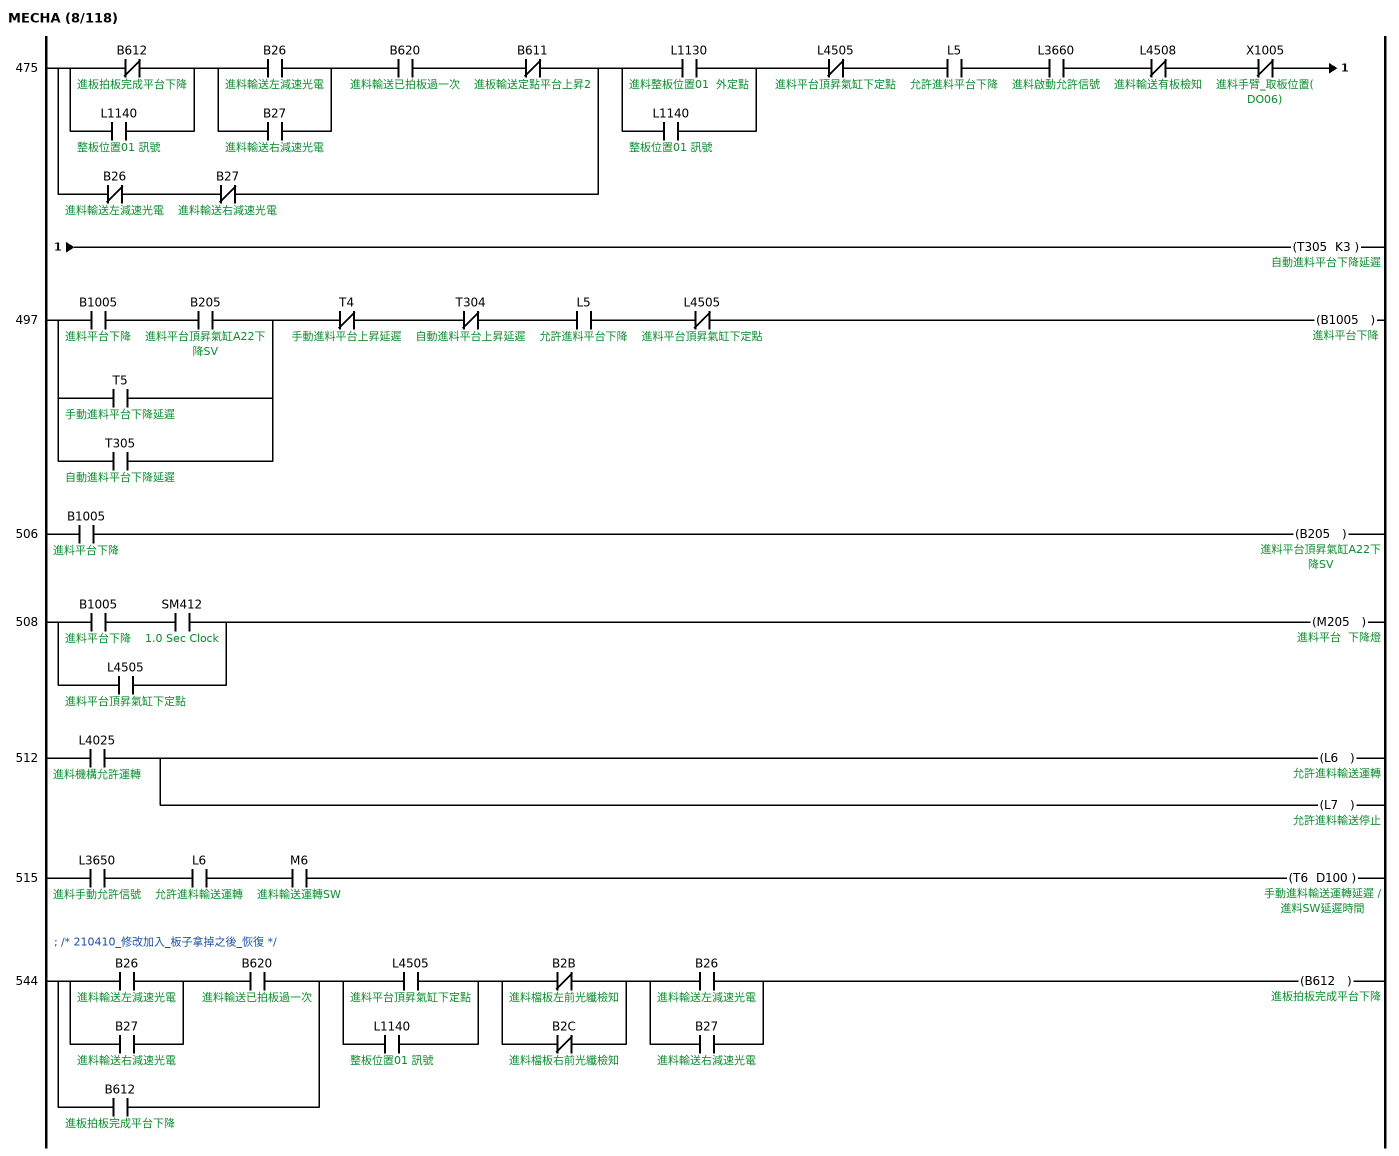
475   LDI     B612  ; 進板拍板完成平台下降
      OR      L1140  ; 整板位置01 訊號
      LD      B26  ; 進料輸送左減速光電
      OR      B27  ; 進料輸送右減速光電
      ANB
      AND     B620  ; 進料輸送已拍板過一次
      ANI     B611  ; 進板輸送定點平台上昇2
      LDI     B26  ; 進料輸送左減速光電
      ANI     B27  ; 進料輸送右減速光電
      ORB
      LD      L1130  ; 進料整板位置01  外定點
      OR      L1140  ; 整板位置01 訊號
      ANB
      ANI     L4505  ; 進料平台頂昇氣缸下定點
      AND     L5  ; 允許進料平台下降
      AND     L3660  ; 進料啟動允許信號
      ANI     L4508  ; 進料輸送有板檢知
      ANI     X1005  ; 進料手臂_取板位置(DO06)
      OUT     T305 K3  ; 自動進料平台下降延遲
497   LD      B1005  ; 進料平台下降
      AND     B205  ; 進料平台頂昇氣缸A22下降SV
      OR      T5  ; 手動進料平台下降延遲
      OR      T305  ; 自動進料平台下降延遲
      ANI     T4  ; 手動進料平台上昇延遲
      ANI     T304  ; 自動進料平台上昇延遲
      AND     L5  ; 允許進料平台下降
      ANI     L4505  ; 進料平台頂昇氣缸下定點
      OUT     B1005  ; 進料平台下降
506   LD      B1005  ; 進料平台下降
      OUT     B205  ; 進料平台頂昇氣缸A22下降SV
508   LD      B1005  ; 進料平台下降
      AND     SM412  ; 1.0 Sec Clock
      OR      L4505  ; 進料平台頂昇氣缸下定點
      OUT     M205  ; 進料平台  下降燈
512   LD      L4025  ; 進料機構允許運轉
      OUT     L6  ; 允許進料輸送運轉
      OUT     L7  ; 允許進料輸送停止
515   LD      L3650  ; 進料手動允許信號
      AND     L6  ; 允許進料輸送運轉
      AND     M6  ; 進料輸送運轉SW
      OUT     T6 D100  ; 手動進料輸送運轉延遲 / 進料SW延遲時間
; /* 210410_修改加入_板子拿掉之後_恢復 */
544   LD      B26  ; 進料輸送左減速光電
      OR      B27  ; 進料輸送右減速光電
      AND     B620  ; 進料輸送已拍板過一次
      OR      B612  ; 進板拍板完成平台下降
      LD      L4505  ; 進料平台頂昇氣缸下定點
      OR      L1140  ; 整板位置01 訊號
      ANB
      LDI     B2B  ; 進料檔板左前光纖檢知
      ORI     B2C  ; 進料檔板右前光纖檢知
      ANB
      LD      B26  ; 進料輸送左減速光電
      OR      B27  ; 進料輸送右減速光電
      ANB
      OUT     B612  ; 進板拍板完成平台下降
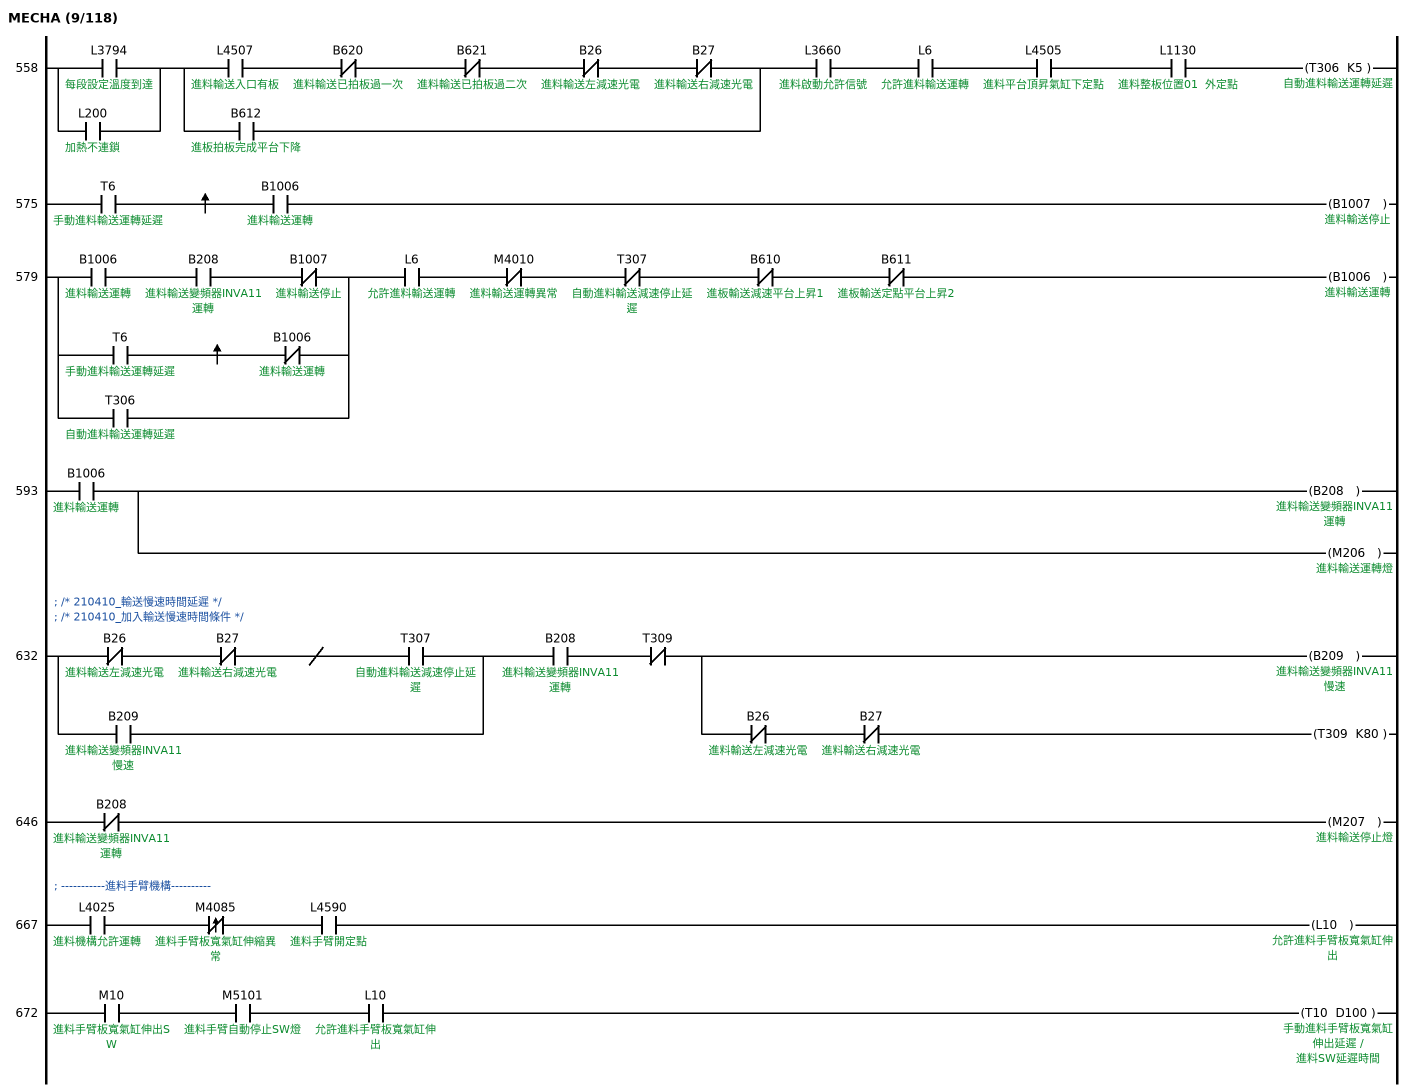
558   LD      L3794  ; 每段設定溫度到達
      OR      L200  ; 加熱不連鎖
      LD      L4507  ; 進料輸送入口有板
      ANI     B620  ; 進料輸送已拍板過一次
      ANI     B621  ; 進料輸送已拍板過二次
      ANI     B26  ; 進料輸送左減速光電
      ANI     B27  ; 進料輸送右減速光電
      OR      B612  ; 進板拍板完成平台下降
      ANB
      AND     L3660  ; 進料啟動允許信號
      AND     L6  ; 允許進料輸送運轉
      AND     L4505  ; 進料平台頂昇氣缸下定點
      AND     L1130  ; 進料整板位置01  外定點
      OUT     T306 K5  ; 自動進料輸送運轉延遲
575   LD      T6  ; 手動進料輸送運轉延遲
      MEP
      AND     B1006  ; 進料輸送運轉
      OUT     B1007  ; 進料輸送停止
579   LD      B1006  ; 進料輸送運轉
      AND     B208  ; 進料輸送變頻器INVA11運轉
      ANI     B1007  ; 進料輸送停止
      LD      T6  ; 手動進料輸送運轉延遲
      MEP
      ANI     B1006  ; 進料輸送運轉
      ORB
      OR      T306  ; 自動進料輸送運轉延遲
      AND     L6  ; 允許進料輸送運轉
      ANI     M4010  ; 進料輸送運轉異常
      ANI     T307  ; 自動進料輸送減速停止延遲
      ANI     B610  ; 進板輸送減速平台上昇1
      ANI     B611  ; 進板輸送定點平台上昇2
      OUT     B1006  ; 進料輸送運轉
593   LD      B1006  ; 進料輸送運轉
      OUT     B208  ; 進料輸送變頻器INVA11運轉
      OUT     M206  ; 進料輸送運轉燈
; /* 210410_輸送慢速時間延遲 */
; /* 210410_加入輸送慢速時間條件 */
632   LDI     B26  ; 進料輸送左減速光電
      ANI     B27  ; 進料輸送右減速光電
      INV
      AND     T307  ; 自動進料輸送減速停止延遲
      OR      B209  ; 進料輸送變頻器INVA11慢速
      AND     B208  ; 進料輸送變頻器INVA11運轉
      ANI     T309
      OUT     B209  ; 進料輸送變頻器INVA11慢速
      ANI     B26  ; 進料輸送左減速光電
      ANI     B27  ; 進料輸送右減速光電
      OUT     T309 K80
646   LDI     B208  ; 進料輸送變頻器INVA11運轉
      OUT     M207  ; 進料輸送停止燈
; -----------進料手臂機構----------
667   LD      L4025  ; 進料機構允許運轉
      ANDPI   M4085  ; 進料手臂板寬氣缸伸縮異常
      AND     L4590  ; 進料手臂開定點
      OUT     L10  ; 允許進料手臂板寬氣缸伸出
672   LD      M10  ; 進料手臂板寬氣缸伸出SW
      AND     M5101  ; 進料手臂自動停止SW燈
      AND     L10  ; 允許進料手臂板寬氣缸伸出
      OUT     T10 D100  ; 手動進料手臂板寬氣缸伸出延遲 / 進料SW延遲時間
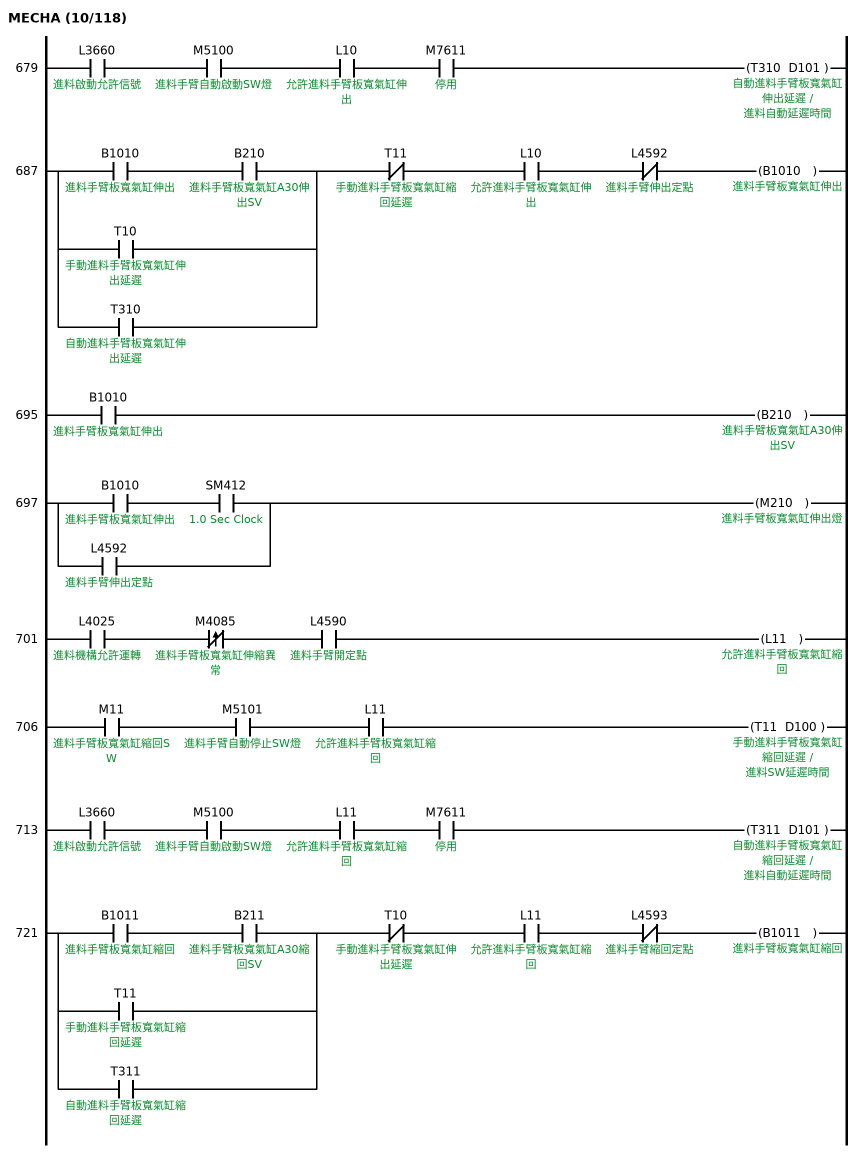
679   LD      L3660  ; 進料啟動允許信號
      AND     M5100  ; 進料手臂自動啟動SW燈
      AND     L10  ; 允許進料手臂板寬氣缸伸出
      AND     M7611  ; 停用
      OUT     T310 D101  ; 自動進料手臂板寬氣缸伸出延遲 / 進料自動延遲時間
687   LD      B1010  ; 進料手臂板寬氣缸伸出
      AND     B210  ; 進料手臂板寬氣缸A30伸出SV
      OR      T10  ; 手動進料手臂板寬氣缸伸出延遲
      OR      T310  ; 自動進料手臂板寬氣缸伸出延遲
      ANI     T11  ; 手動進料手臂板寬氣缸縮回延遲
      AND     L10  ; 允許進料手臂板寬氣缸伸出
      ANI     L4592  ; 進料手臂伸出定點
      OUT     B1010  ; 進料手臂板寬氣缸伸出
695   LD      B1010  ; 進料手臂板寬氣缸伸出
      OUT     B210  ; 進料手臂板寬氣缸A30伸出SV
697   LD      B1010  ; 進料手臂板寬氣缸伸出
      AND     SM412  ; 1.0 Sec Clock
      OR      L4592  ; 進料手臂伸出定點
      OUT     M210  ; 進料手臂板寬氣缸伸出燈
701   LD      L4025  ; 進料機構允許運轉
      ANDPI   M4085  ; 進料手臂板寬氣缸伸縮異常
      AND     L4590  ; 進料手臂開定點
      OUT     L11  ; 允許進料手臂板寬氣缸縮回
706   LD      M11  ; 進料手臂板寬氣缸縮回SW
      AND     M5101  ; 進料手臂自動停止SW燈
      AND     L11  ; 允許進料手臂板寬氣缸縮回
      OUT     T11 D100  ; 手動進料手臂板寬氣缸縮回延遲 / 進料SW延遲時間
713   LD      L3660  ; 進料啟動允許信號
      AND     M5100  ; 進料手臂自動啟動SW燈
      AND     L11  ; 允許進料手臂板寬氣缸縮回
      AND     M7611  ; 停用
      OUT     T311 D101  ; 自動進料手臂板寬氣缸縮回延遲 / 進料自動延遲時間
721   LD      B1011  ; 進料手臂板寬氣缸縮回
      AND     B211  ; 進料手臂板寬氣缸A30縮回SV
      OR      T11  ; 手動進料手臂板寬氣缸縮回延遲
      OR      T311  ; 自動進料手臂板寬氣缸縮回延遲
      ANI     T10  ; 手動進料手臂板寬氣缸伸出延遲
      AND     L11  ; 允許進料手臂板寬氣缸縮回
      ANI     L4593  ; 進料手臂縮回定點
      OUT     B1011  ; 進料手臂板寬氣缸縮回
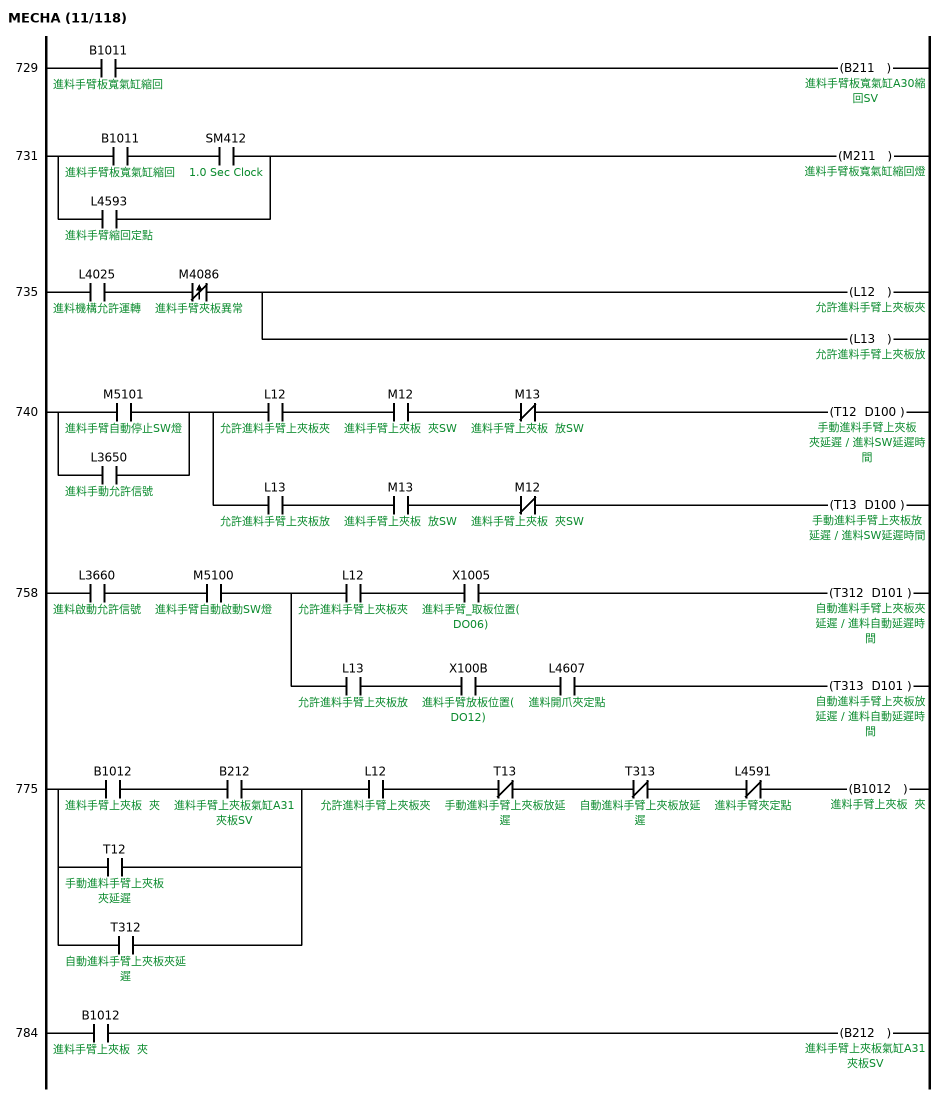
729   LD      B1011  ; 進料手臂板寬氣缸縮回
      OUT     B211  ; 進料手臂板寬氣缸A30縮回SV
731   LD      B1011  ; 進料手臂板寬氣缸縮回
      AND     SM412  ; 1.0 Sec Clock
      OR      L4593  ; 進料手臂縮回定點
      OUT     M211  ; 進料手臂板寬氣缸縮回燈
735   LD      L4025  ; 進料機構允許運轉
      ANDPI   M4086  ; 進料手臂夾板異常
      OUT     L12  ; 允許進料手臂上夾板夾
      OUT     L13  ; 允許進料手臂上夾板放
740   LD      M5101  ; 進料手臂自動停止SW燈
      OR      L3650  ; 進料手動允許信號
      MPS
      AND     L12  ; 允許進料手臂上夾板夾
      AND     M12  ; 進料手臂上夾板  夾SW
      ANI     M13  ; 進料手臂上夾板  放SW
      OUT     T12 D100  ; 手動進料手臂上夾板  夾延遲 / 進料SW延遲時間
      MPP
      AND     L13  ; 允許進料手臂上夾板放
      AND     M13  ; 進料手臂上夾板  放SW
      ANI     M12  ; 進料手臂上夾板  夾SW
      OUT     T13 D100  ; 手動進料手臂上夾板放延遲 / 進料SW延遲時間
758   LD      L3660  ; 進料啟動允許信號
      AND     M5100  ; 進料手臂自動啟動SW燈
      MPS
      AND     L12  ; 允許進料手臂上夾板夾
      AND     X1005  ; 進料手臂_取板位置(DO06)
      OUT     T312 D101  ; 自動進料手臂上夾板夾延遲 / 進料自動延遲時間
      MPP
      AND     L13  ; 允許進料手臂上夾板放
      AND     X100B  ; 進料手臂放板位置(DO12)
      AND     L4607  ; 進料開爪夾定點
      OUT     T313 D101  ; 自動進料手臂上夾板放延遲 / 進料自動延遲時間
775   LD      B1012  ; 進料手臂上夾板  夾
      AND     B212  ; 進料手臂上夾板氣缸A31夾板SV
      OR      T12  ; 手動進料手臂上夾板  夾延遲
      OR      T312  ; 自動進料手臂上夾板夾延遲
      AND     L12  ; 允許進料手臂上夾板夾
      ANI     T13  ; 手動進料手臂上夾板放延遲
      ANI     T313  ; 自動進料手臂上夾板放延遲
      ANI     L4591  ; 進料手臂夾定點
      OUT     B1012  ; 進料手臂上夾板  夾
784   LD      B1012  ; 進料手臂上夾板  夾
      OUT     B212  ; 進料手臂上夾板氣缸A31夾板SV
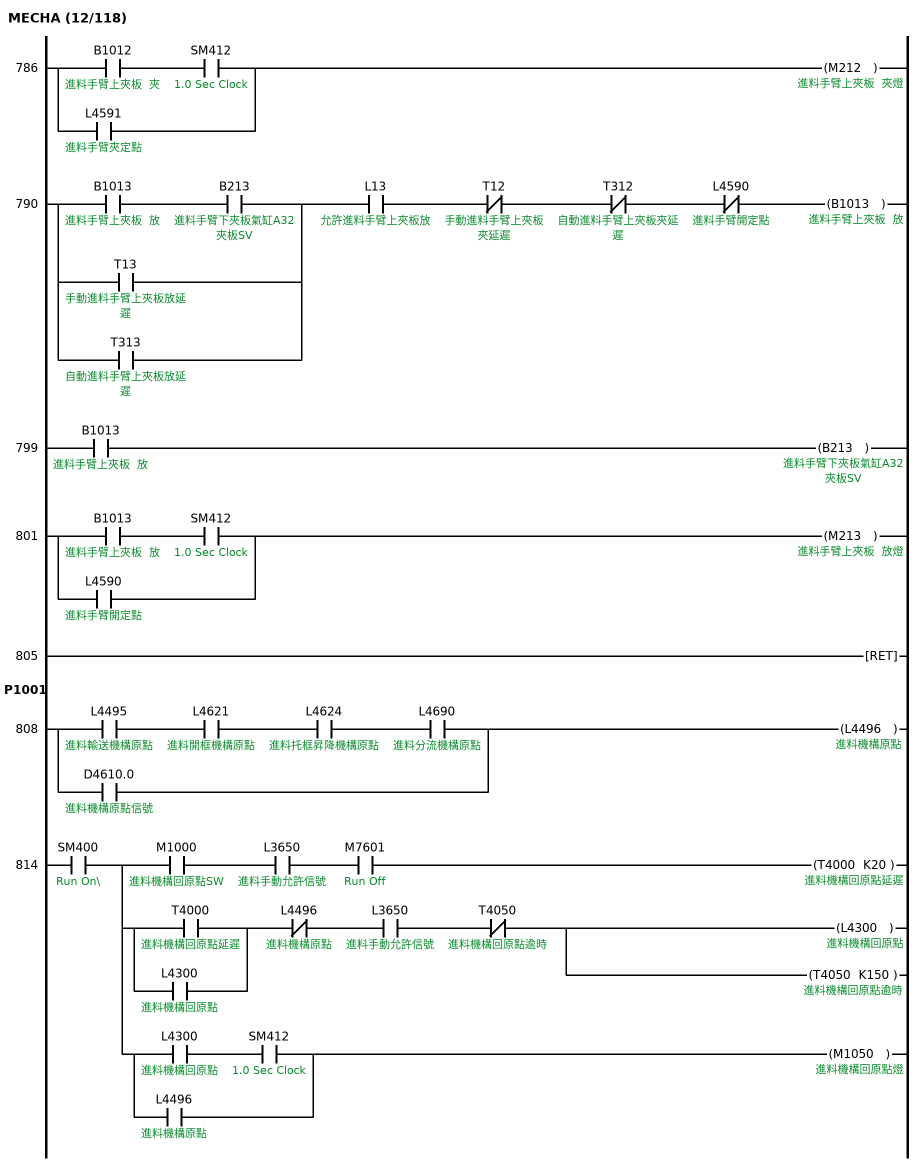
786   LD      B1012  ; 進料手臂上夾板  夾
      AND     SM412  ; 1.0 Sec Clock
      OR      L4591  ; 進料手臂夾定點
      OUT     M212  ; 進料手臂上夾板  夾燈
790   LD      B1013  ; 進料手臂上夾板  放
      AND     B213  ; 進料手臂下夾板氣缸A32夾板SV
      OR      T13  ; 手動進料手臂上夾板放延遲
      OR      T313  ; 自動進料手臂上夾板放延遲
      AND     L13  ; 允許進料手臂上夾板放
      ANI     T12  ; 手動進料手臂上夾板  夾延遲
      ANI     T312  ; 自動進料手臂上夾板夾延遲
      ANI     L4590  ; 進料手臂開定點
      OUT     B1013  ; 進料手臂上夾板  放
799   LD      B1013  ; 進料手臂上夾板  放
      OUT     B213  ; 進料手臂下夾板氣缸A32夾板SV
801   LD      B1013  ; 進料手臂上夾板  放
      AND     SM412  ; 1.0 Sec Clock
      OR      L4590  ; 進料手臂開定點
      OUT     M213  ; 進料手臂上夾板  放燈
805   RET
      P1001
808   LD      L4495  ; 進料輸送機構原點
      AND     L4621  ; 進料開框機構原點
      AND     L4624  ; 進料托框昇降機構原點
      AND     L4690  ; 進料分流機構原點
      OR      D4610.0  ; 進料機構原點信號
      OUT     L4496  ; 進料機構原點
814   LD      SM400  ; Run On\
      MPS
      AND     M1000  ; 進料機構回原點SW
      AND     L3650  ; 進料手動允許信號
      AND     M7601  ; Run Off
      OUT     T4000 K20  ; 進料機構回原點延遲
      MRD
      LD      T4000  ; 進料機構回原點延遲
      OR      L4300  ; 進料機構回原點
      ANB
      ANI     L4496  ; 進料機構原點
      AND     L3650  ; 進料手動允許信號
      ANI     T4050  ; 進料機構回原點逾時
      OUT     L4300  ; 進料機構回原點
      OUT     T4050 K150  ; 進料機構回原點逾時
      MPP
      LD      L4300  ; 進料機構回原點
      AND     SM412  ; 1.0 Sec Clock
      OR      L4496  ; 進料機構原點
      ANB
      OUT     M1050  ; 進料機構回原點燈
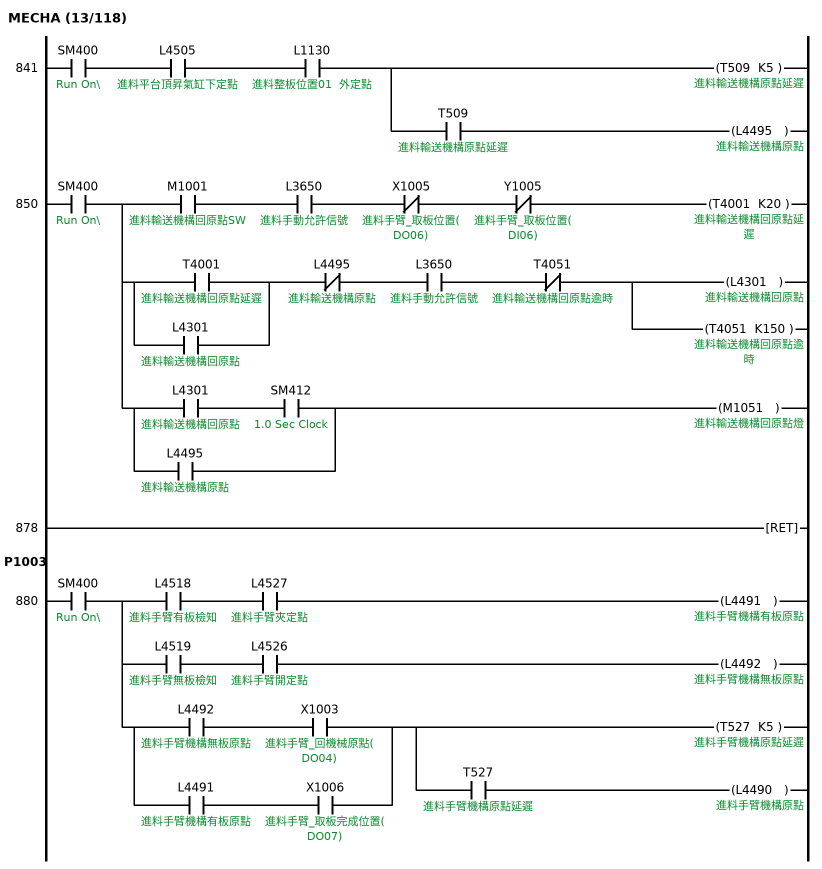
841   LD      SM400  ; Run On\
      AND     L4505  ; 進料平台頂昇氣缸下定點
      AND     L1130  ; 進料整板位置01  外定點
      OUT     T509 K5  ; 進料輸送機構原點延遲
      AND     T509  ; 進料輸送機構原點延遲
      OUT     L4495  ; 進料輸送機構原點
850   LD      SM400  ; Run On\
      MPS
      AND     M1001  ; 進料輸送機構回原點SW
      AND     L3650  ; 進料手動允許信號
      ANI     X1005  ; 進料手臂_取板位置(DO06)
      ANI     Y1005  ; 進料手臂_取板位置(DI06)
      OUT     T4001 K20  ; 進料輸送機構回原點延遲
      MRD
      LD      T4001  ; 進料輸送機構回原點延遲
      OR      L4301  ; 進料輸送機構回原點
      ANB
      ANI     L4495  ; 進料輸送機構原點
      AND     L3650  ; 進料手動允許信號
      ANI     T4051  ; 進料輸送機構回原點逾時
      OUT     L4301  ; 進料輸送機構回原點
      OUT     T4051 K150  ; 進料輸送機構回原點逾時
      MPP
      LD      L4301  ; 進料輸送機構回原點
      AND     SM412  ; 1.0 Sec Clock
      OR      L4495  ; 進料輸送機構原點
      ANB
      OUT     M1051  ; 進料輸送機構回原點燈
878   RET
      P1003
880   LD      SM400  ; Run On\
      MPS
      AND     L4518  ; 進料手臂有板檢知
      AND     L4527  ; 進料手臂夾定點
      OUT     L4491  ; 進料手臂機構有板原點
      MRD
      AND     L4519  ; 進料手臂無板檢知
      AND     L4526  ; 進料手臂開定點
      OUT     L4492  ; 進料手臂機構無板原點
      MPP
      LD      L4492  ; 進料手臂機構無板原點
      AND     X1003  ; 進料手臂_回機械原點(DO04)
      LD      L4491  ; 進料手臂機構有板原點
      AND     X1006  ; 進料手臂_取板完成位置(DO07)
      ORB
      ANB
      OUT     T527 K5  ; 進料手臂機構原點延遲
      AND     T527  ; 進料手臂機構原點延遲
      OUT     L4490  ; 進料手臂機構原點
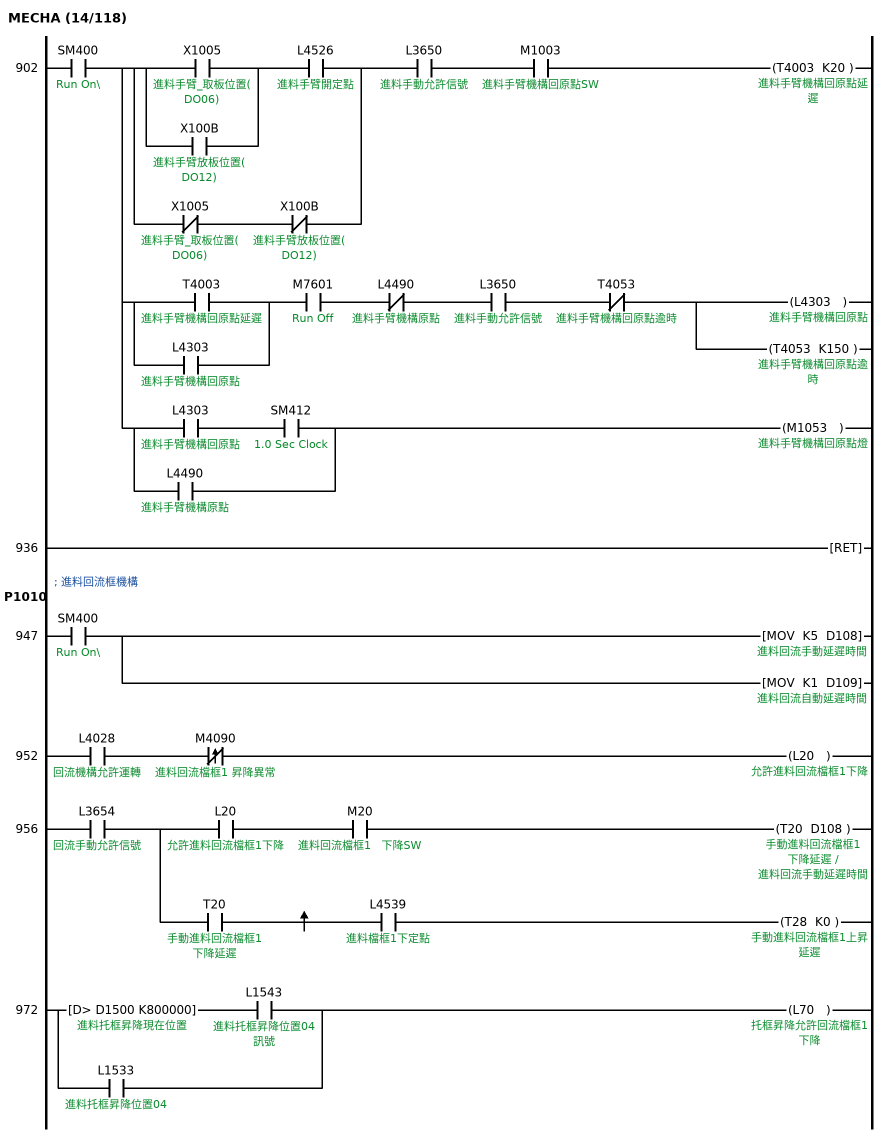
902   LD      SM400  ; Run On\
      MPS
      LD      X1005  ; 進料手臂_取板位置(DO06)
      OR      X100B  ; 進料手臂放板位置(DO12)
      AND     L4526  ; 進料手臂開定點
      LDI     X1005  ; 進料手臂_取板位置(DO06)
      ANI     X100B  ; 進料手臂放板位置(DO12)
      ORB
      ANB
      AND     L3650  ; 進料手動允許信號
      AND     M1003  ; 進料手臂機構回原點SW
      OUT     T4003 K20  ; 進料手臂機構回原點延遲
      MRD
      LD      T4003  ; 進料手臂機構回原點延遲
      OR      L4303  ; 進料手臂機構回原點
      ANB
      AND     M7601  ; Run Off
      ANI     L4490  ; 進料手臂機構原點
      AND     L3650  ; 進料手動允許信號
      ANI     T4053  ; 進料手臂機構回原點逾時
      OUT     L4303  ; 進料手臂機構回原點
      OUT     T4053 K150  ; 進料手臂機構回原點逾時
      MPP
      LD      L4303  ; 進料手臂機構回原點
      AND     SM412  ; 1.0 Sec Clock
      OR      L4490  ; 進料手臂機構原點
      ANB
      OUT     M1053  ; 進料手臂機構回原點燈
936   RET
; 進料回流框機構
      P1010
947   LD      SM400  ; Run On\
      MOV     K5 D108  ; 進料回流手動延遲時間
      MOV     K1 D109  ; 進料回流自動延遲時間
952   LD      L4028  ; 回流機構允許運轉
      ANDPI   M4090  ; 進料回流檔框1 昇降異常
      OUT     L20  ; 允許進料回流檔框1下降
956   LD      L3654  ; 回流手動允許信號
      MPS
      AND     L20  ; 允許進料回流檔框1下降
      AND     M20  ; 進料回流檔框1   下降SW
      OUT     T20 D108  ; 手動進料回流檔框1   下降延遲 / 進料回流手動延遲時間
      MPP
      AND     T20  ; 手動進料回流檔框1   下降延遲
      MEP
      AND     L4539  ; 進料檔框1下定點
      OUT     T28 K0  ; 手動進料回流檔框1上昇延遲
972   LDD>    D1500 K800000  ; 進料托框昇降現在位置
      AND     L1543  ; 進料托框昇降位置04 訊號
      OR      L1533  ; 進料托框昇降位置04
      OUT     L70  ; 托框昇降允許回流檔框1下降
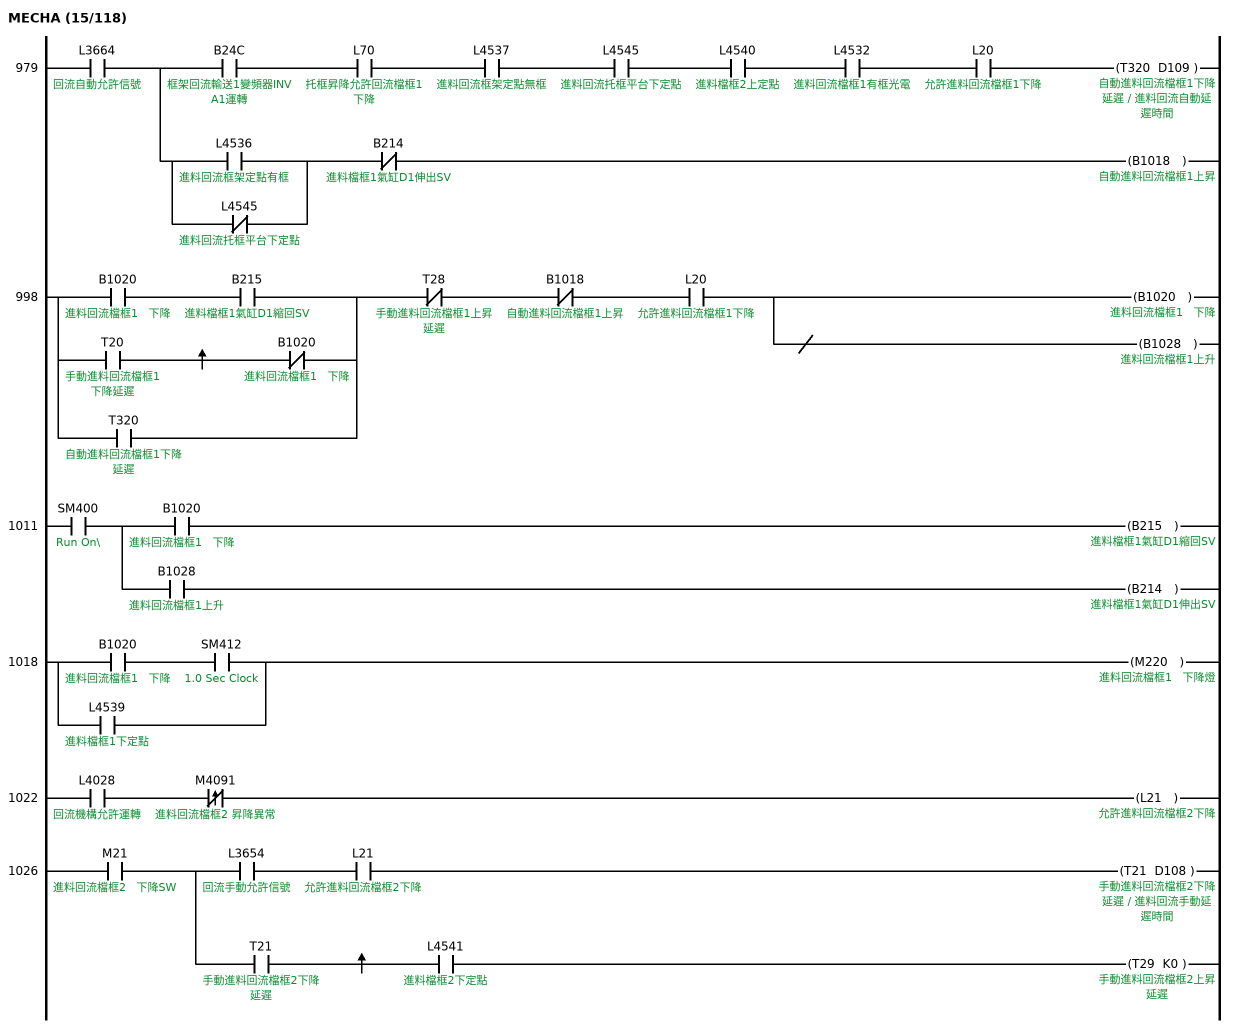
979   LD      L3664  ; 回流自動允許信號
      MPS
      AND     B24C  ; 框架回流輸送1變頻器INVA1運轉
      AND     L70  ; 托框昇降允許回流檔框1下降
      AND     L4537  ; 進料回流框架定點無框
      AND     L4545  ; 進料回流托框平台下定點
      AND     L4540  ; 進料檔框2上定點
      AND     L4532  ; 進料回流檔框1有框光電
      AND     L20  ; 允許進料回流檔框1下降
      OUT     T320 D109  ; 自動進料回流檔框1下降延遲 / 進料回流自動延遲時間
      MPP
      LD      L4536  ; 進料回流框架定點有框
      ORI     L4545  ; 進料回流托框平台下定點
      ANB
      ANI     B214  ; 進料檔框1氣缸D1伸出SV
      OUT     B1018  ; 自動進料回流檔框1上昇
998   LD      B1020  ; 進料回流檔框1   下降
      AND     B215  ; 進料檔框1氣缸D1縮回SV
      LD      T20  ; 手動進料回流檔框1   下降延遲
      MEP
      ANI     B1020  ; 進料回流檔框1   下降
      ORB
      OR      T320  ; 自動進料回流檔框1下降延遲
      ANI     T28  ; 手動進料回流檔框1上昇延遲
      ANI     B1018  ; 自動進料回流檔框1上昇
      AND     L20  ; 允許進料回流檔框1下降
      OUT     B1020  ; 進料回流檔框1   下降
      INV
      OUT     B1028  ; 進料回流檔框1上升
1011  LD      SM400  ; Run On\
      MPS
      AND     B1020  ; 進料回流檔框1   下降
      OUT     B215  ; 進料檔框1氣缸D1縮回SV
      MPP
      AND     B1028  ; 進料回流檔框1上升
      OUT     B214  ; 進料檔框1氣缸D1伸出SV
1018  LD      B1020  ; 進料回流檔框1   下降
      AND     SM412  ; 1.0 Sec Clock
      OR      L4539  ; 進料檔框1下定點
      OUT     M220  ; 進料回流檔框1   下降燈
1022  LD      L4028  ; 回流機構允許運轉
      ANDPI   M4091  ; 進料回流檔框2 昇降異常
      OUT     L21  ; 允許進料回流檔框2下降
1026  LD      M21  ; 進料回流檔框2   下降SW
      MPS
      AND     L3654  ; 回流手動允許信號
      AND     L21  ; 允許進料回流檔框2下降
      OUT     T21 D108  ; 手動進料回流檔框2下降延遲 / 進料回流手動延遲時間
      MPP
      AND     T21  ; 手動進料回流檔框2下降延遲
      MEP
      AND     L4541  ; 進料檔框2下定點
      OUT     T29 K0  ; 手動進料回流檔框2上昇延遲
